
FUNCTION "FC_AI_MAPPING" : VOID
TITLE =
VERSION : 0.1


VAR_TEMP
  PIW512_DI : DINT ;
END_VAR
BEGIN

NETWORK
TITLE =
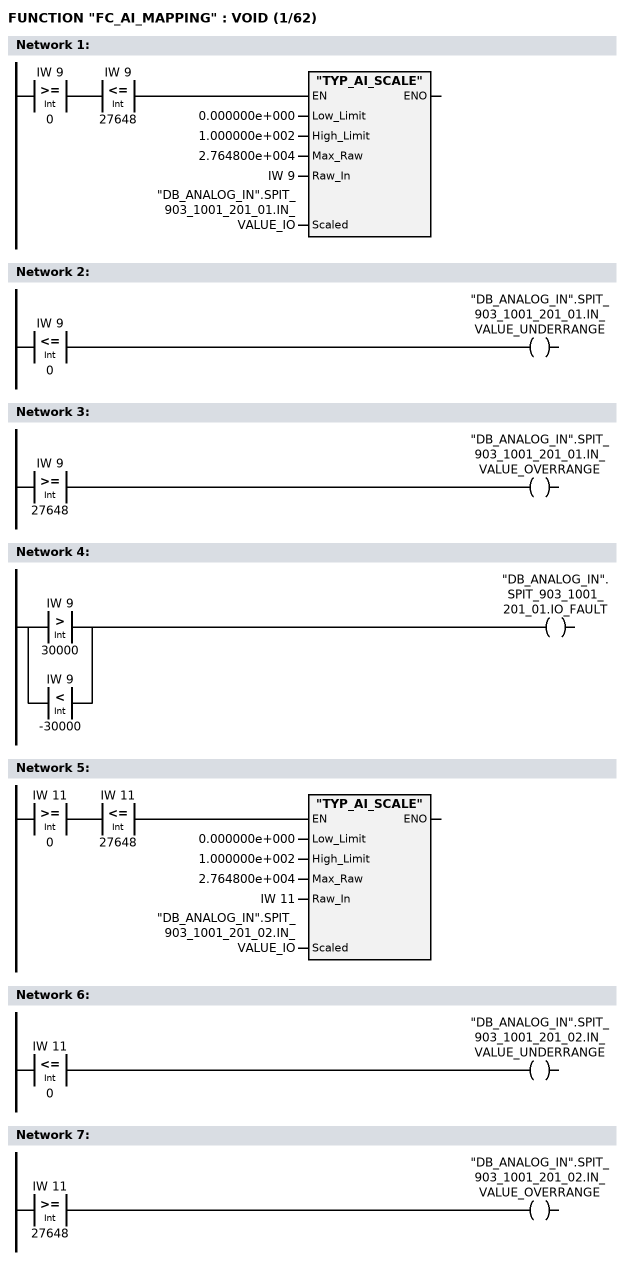

      A(    ;
      L     IW      9;
      L     0;
      >=I   ;
      )     ;
      A(    ;
      L     IW      9;

      L     27648;
      <=I   ;
      )     ;
      JNB   _001;
      CALL "TYP_AI_SCALE" (
           Low_Limit                := 0.000000e+000,
           High_Limit               := 1.000000e+002,
           Max_Raw                  := 2.764800e+004,
           Raw_In                   := IW      9,
           Scaled                   := "DB_ANALOG_IN".SPIT_903_1001_201_01.IN_VALUE_IO);
_001: NOP   0;
NETWORK
TITLE =

      L     IW      9;
      L     0;
      <=I   ;
      =     "DB_ANALOG_IN".SPIT_903_1001_201_01.IN_VALUE_UNDERRANGE;
NETWORK
TITLE =

      L     IW      9;
      L     27648;
      >=I   ;
      =     "DB_ANALOG_IN".SPIT_903_1001_201_01.IN_VALUE_OVERRANGE;
NETWORK
TITLE =

      O(    ;
      L     IW      9;
      L     30000;
      >I    ;
      )     ;
      O(    ;
      L     IW      9;
      L     -30000;
      <I    ;
      )     ;
      =     "DB_ANALOG_IN".SPIT_903_1001_201_01.IO_FAULT;

NETWORK
TITLE =

      A(    ;
      L     IW      11;
      L     0;
      >=I   ;
      )     ;
      A(    ;
      L     IW      11;

      L     27648;
      <=I   ;
      )     ;
      JNB   _002;
      CALL "TYP_AI_SCALE" (
           Low_Limit                := 0.000000e+000,
           High_Limit               := 1.000000e+002,
           Max_Raw                  := 2.764800e+004,
           Raw_In                   := IW      11,
           Scaled                   := "DB_ANALOG_IN".SPIT_903_1001_201_02.IN_VALUE_IO);
_002: NOP   0;
NETWORK
TITLE =

      L     IW      11;
      L     0;
      <=I   ;
      =     "DB_ANALOG_IN".SPIT_903_1001_201_02.IN_VALUE_UNDERRANGE;
NETWORK
TITLE =

      L     IW      11;
      L     27648;
      >=I   ;
      =     "DB_ANALOG_IN".SPIT_903_1001_201_02.IN_VALUE_OVERRANGE;
NETWORK
TITLE =
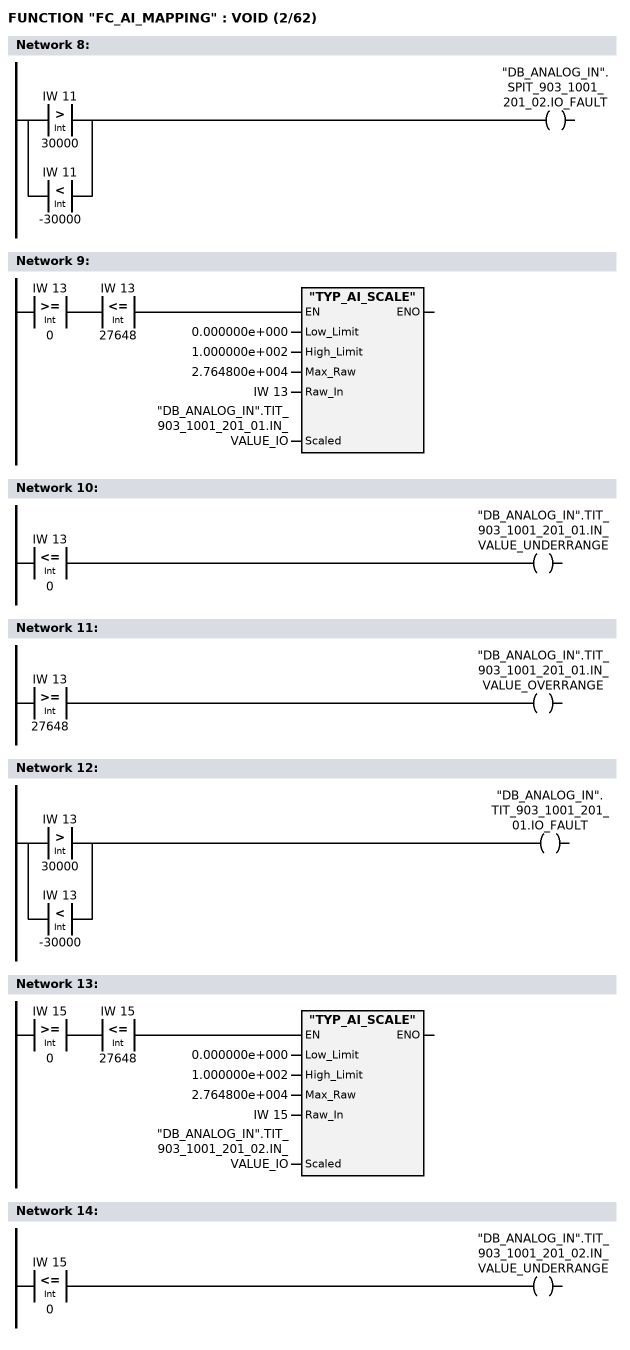

      O(    ;
      L     IW      11;
      L     30000;
      >I    ;
      )     ;
      O(    ;
      L     IW      11;
      L     -30000;
      <I    ;
      )     ;
      =     "DB_ANALOG_IN".SPIT_903_1001_201_02.IO_FAULT;

NETWORK
TITLE =

      A(    ;
      L     IW      13;
      L     0;
      >=I   ;
      )     ;
      A(    ;
      L     IW      13;

      L     27648;
      <=I   ;
      )     ;
      JNB   _003;
      CALL "TYP_AI_SCALE" (
           Low_Limit                := 0.000000e+000,
           High_Limit               := 1.000000e+002,
           Max_Raw                  := 2.764800e+004,
           Raw_In                   := IW      13,
           Scaled                   := "DB_ANALOG_IN".TIT_903_1001_201_01.IN_VALUE_IO);
_003: NOP   0;
NETWORK
TITLE =

      L     IW      13;
      L     0;
      <=I   ;
      =     "DB_ANALOG_IN".TIT_903_1001_201_01.IN_VALUE_UNDERRANGE;
NETWORK
TITLE =

      L     IW      13;
      L     27648;
      >=I   ;
      =     "DB_ANALOG_IN".TIT_903_1001_201_01.IN_VALUE_OVERRANGE;
NETWORK
TITLE =

      O(    ;
      L     IW      13;
      L     30000;
      >I    ;
      )     ;
      O(    ;
      L     IW      13;
      L     -30000;
      <I    ;
      )     ;
      =     "DB_ANALOG_IN".TIT_903_1001_201_01.IO_FAULT;

NETWORK
TITLE =

      A(    ;
      L     IW      15;
      L     0;
      >=I   ;
      )     ;
      A(    ;
      L     IW      15;

      L     27648;
      <=I   ;
      )     ;
      JNB   _004;
      CALL "TYP_AI_SCALE" (
           Low_Limit                := 0.000000e+000,
           High_Limit               := 1.000000e+002,
           Max_Raw                  := 2.764800e+004,
           Raw_In                   := IW      15,
           Scaled                   := "DB_ANALOG_IN".TIT_903_1001_201_02.IN_VALUE_IO);
_004: NOP   0;
NETWORK
TITLE =

      L     IW      15;
      L     0;
      <=I   ;
      =     "DB_ANALOG_IN".TIT_903_1001_201_02.IN_VALUE_UNDERRANGE;
NETWORK
TITLE =
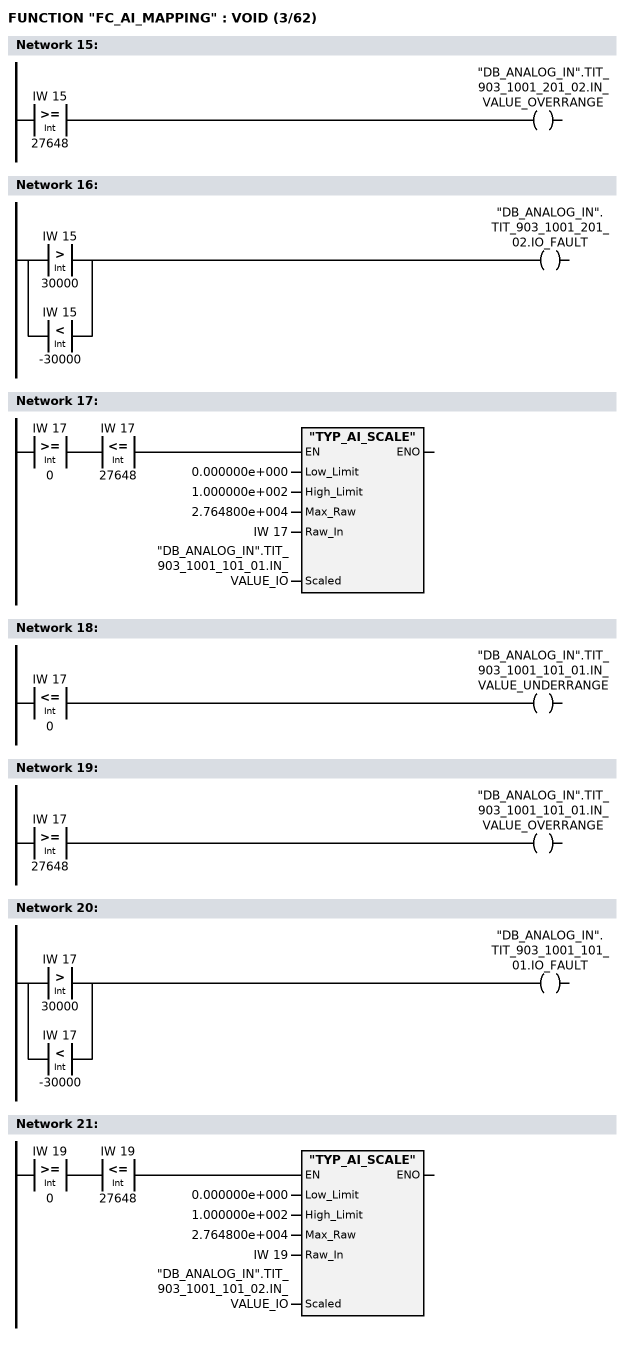

      L     IW      15;
      L     27648;
      >=I   ;
      =     "DB_ANALOG_IN".TIT_903_1001_201_02.IN_VALUE_OVERRANGE;
NETWORK
TITLE =

      O(    ;
      L     IW      15;
      L     30000;
      >I    ;
      )     ;
      O(    ;
      L     IW      15;
      L     -30000;
      <I    ;
      )     ;
      =     "DB_ANALOG_IN".TIT_903_1001_201_02.IO_FAULT;

NETWORK
TITLE =

      A(    ;
      L     IW      17;
      L     0;
      >=I   ;
      )     ;
      A(    ;
      L     IW      17;

      L     27648;
      <=I   ;
      )     ;
      JNB   _005;
      CALL "TYP_AI_SCALE" (
           Low_Limit                := 0.000000e+000,
           High_Limit               := 1.000000e+002,
           Max_Raw                  := 2.764800e+004,
           Raw_In                   := IW      17,
           Scaled                   := "DB_ANALOG_IN".TIT_903_1001_101_01.IN_VALUE_IO);
_005: NOP   0;
NETWORK
TITLE =

      L     IW      17;
      L     0;
      <=I   ;
      =     "DB_ANALOG_IN".TIT_903_1001_101_01.IN_VALUE_UNDERRANGE;
NETWORK
TITLE =

      L     IW      17;
      L     27648;
      >=I   ;
      =     "DB_ANALOG_IN".TIT_903_1001_101_01.IN_VALUE_OVERRANGE;
NETWORK
TITLE =

      O(    ;
      L     IW      17;
      L     30000;
      >I    ;
      )     ;
      O(    ;
      L     IW      17;
      L     -30000;
      <I    ;
      )     ;
      =     "DB_ANALOG_IN".TIT_903_1001_101_01.IO_FAULT;

NETWORK
TITLE =

      A(    ;
      L     IW      19;
      L     0;
      >=I   ;
      )     ;
      A(    ;
      L     IW      19;

      L     27648;
      <=I   ;
      )     ;
      JNB   _006;
      CALL "TYP_AI_SCALE" (
           Low_Limit                := 0.000000e+000,
           High_Limit               := 1.000000e+002,
           Max_Raw                  := 2.764800e+004,
           Raw_In                   := IW      19,
           Scaled                   := "DB_ANALOG_IN".TIT_903_1001_101_02.IN_VALUE_IO);
_006: NOP   0;
NETWORK
TITLE =
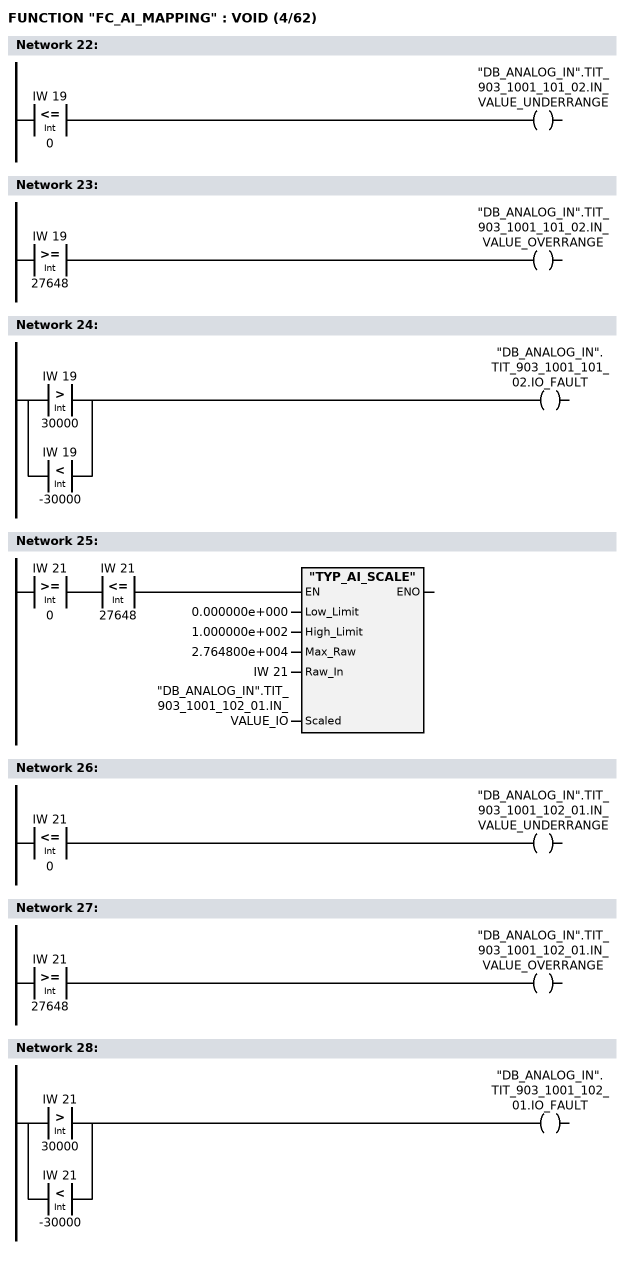

      L     IW      19;
      L     0;
      <=I   ;
      =     "DB_ANALOG_IN".TIT_903_1001_101_02.IN_VALUE_UNDERRANGE;
NETWORK
TITLE =

      L     IW      19;
      L     27648;
      >=I   ;
      =     "DB_ANALOG_IN".TIT_903_1001_101_02.IN_VALUE_OVERRANGE;
NETWORK
TITLE =

      O(    ;
      L     IW      19;
      L     30000;
      >I    ;
      )     ;
      O(    ;
      L     IW      19;
      L     -30000;
      <I    ;
      )     ;
      =     "DB_ANALOG_IN".TIT_903_1001_101_02.IO_FAULT;

NETWORK
TITLE =

      A(    ;
      L     IW      21;
      L     0;
      >=I   ;
      )     ;
      A(    ;
      L     IW      21;

      L     27648;
      <=I   ;
      )     ;
      JNB   _007;
      CALL "TYP_AI_SCALE" (
           Low_Limit                := 0.000000e+000,
           High_Limit               := 1.000000e+002,
           Max_Raw                  := 2.764800e+004,
           Raw_In                   := IW      21,
           Scaled                   := "DB_ANALOG_IN".TIT_903_1001_102_01.IN_VALUE_IO);
_007: NOP   0;
NETWORK
TITLE =

      L     IW      21;
      L     0;
      <=I   ;
      =     "DB_ANALOG_IN".TIT_903_1001_102_01.IN_VALUE_UNDERRANGE;
NETWORK
TITLE =

      L     IW      21;
      L     27648;
      >=I   ;
      =     "DB_ANALOG_IN".TIT_903_1001_102_01.IN_VALUE_OVERRANGE;
NETWORK
TITLE =

      O(    ;
      L     IW      21;
      L     30000;
      >I    ;
      )     ;
      O(    ;
      L     IW      21;
      L     -30000;
      <I    ;
      )     ;
      =     "DB_ANALOG_IN".TIT_903_1001_102_01.IO_FAULT;

NETWORK
TITLE =
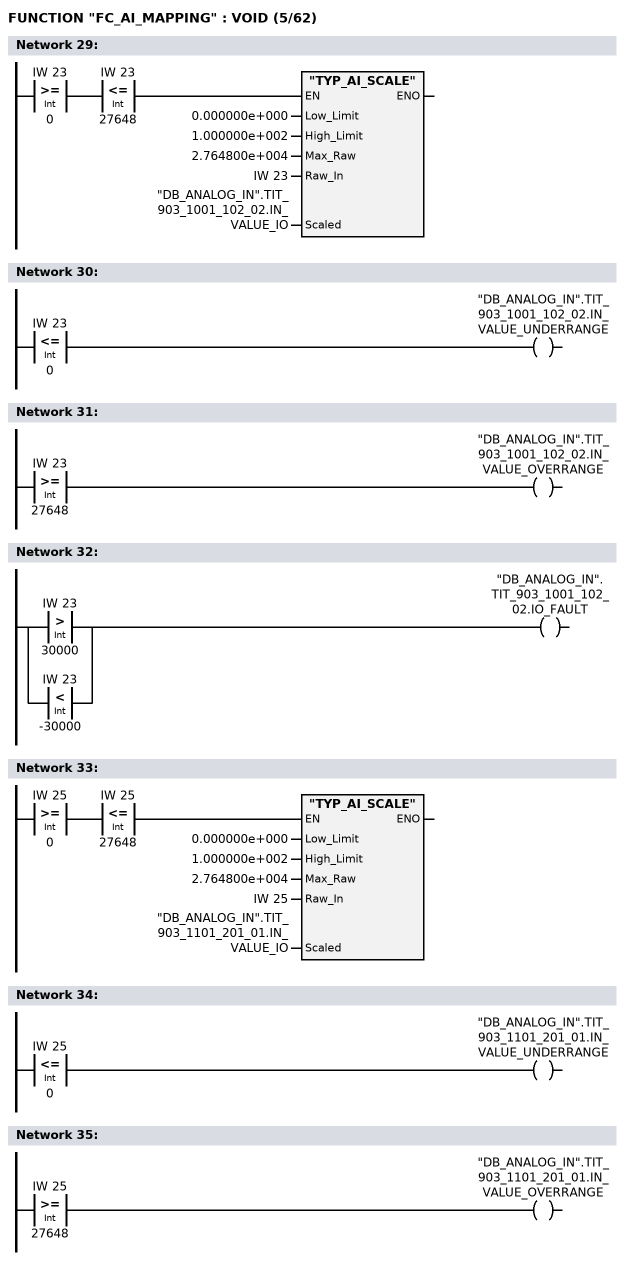

      A(    ;
      L     IW      23;
      L     0;
      >=I   ;
      )     ;
      A(    ;
      L     IW      23;

      L     27648;
      <=I   ;
      )     ;
      JNB   _008;
      CALL "TYP_AI_SCALE" (
           Low_Limit                := 0.000000e+000,
           High_Limit               := 1.000000e+002,
           Max_Raw                  := 2.764800e+004,
           Raw_In                   := IW      23,
           Scaled                   := "DB_ANALOG_IN".TIT_903_1001_102_02.IN_VALUE_IO);
_008: NOP   0;
NETWORK
TITLE =

      L     IW      23;
      L     0;
      <=I   ;
      =     "DB_ANALOG_IN".TIT_903_1001_102_02.IN_VALUE_UNDERRANGE;
NETWORK
TITLE =

      L     IW      23;
      L     27648;
      >=I   ;
      =     "DB_ANALOG_IN".TIT_903_1001_102_02.IN_VALUE_OVERRANGE;
NETWORK
TITLE =

      O(    ;
      L     IW      23;
      L     30000;
      >I    ;
      )     ;
      O(    ;
      L     IW      23;
      L     -30000;
      <I    ;
      )     ;
      =     "DB_ANALOG_IN".TIT_903_1001_102_02.IO_FAULT;

NETWORK
TITLE =

      A(    ;
      L     IW      25;
      L     0;
      >=I   ;
      )     ;
      A(    ;
      L     IW      25;

      L     27648;
      <=I   ;
      )     ;
      JNB   _009;
      CALL "TYP_AI_SCALE" (
           Low_Limit                := 0.000000e+000,
           High_Limit               := 1.000000e+002,
           Max_Raw                  := 2.764800e+004,
           Raw_In                   := IW      25,
           Scaled                   := "DB_ANALOG_IN".TIT_903_1101_201_01.IN_VALUE_IO);
_009: NOP   0;
NETWORK
TITLE =

      L     IW      25;
      L     0;
      <=I   ;
      =     "DB_ANALOG_IN".TIT_903_1101_201_01.IN_VALUE_UNDERRANGE;
NETWORK
TITLE =

      L     IW      25;
      L     27648;
      >=I   ;
      =     "DB_ANALOG_IN".TIT_903_1101_201_01.IN_VALUE_OVERRANGE;
NETWORK
TITLE =
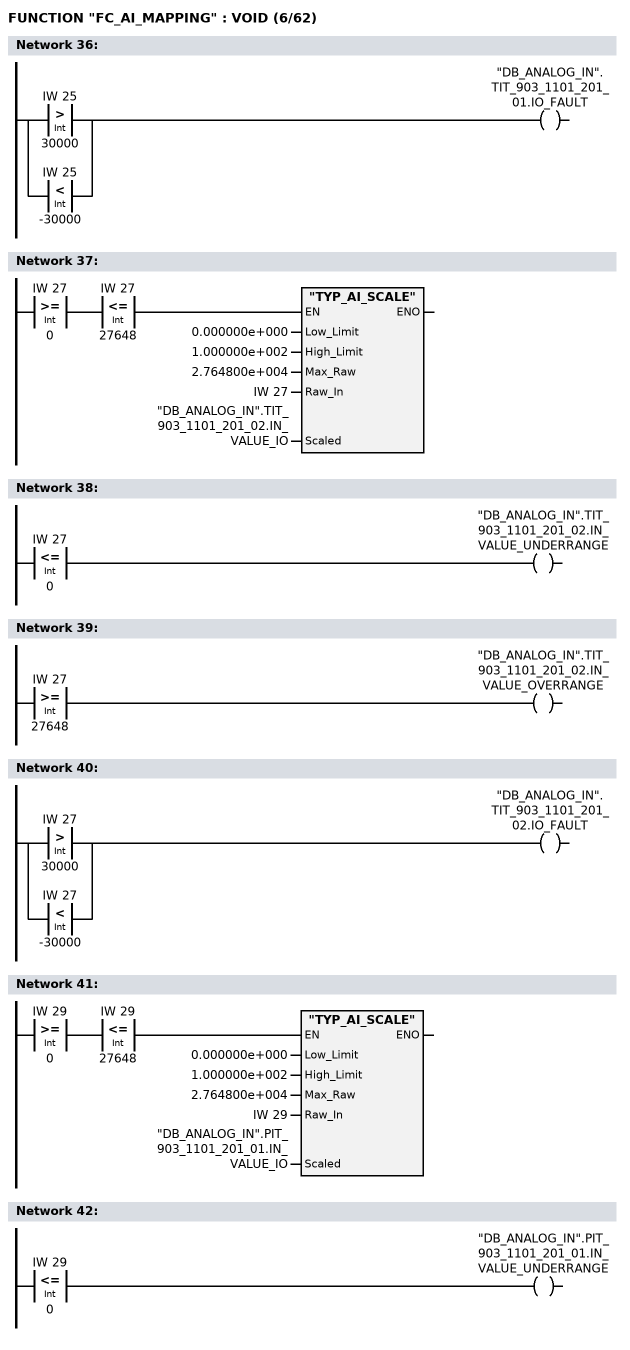

      O(    ;
      L     IW      25;
      L     30000;
      >I    ;
      )     ;
      O(    ;
      L     IW      25;
      L     -30000;
      <I    ;
      )     ;
      =     "DB_ANALOG_IN".TIT_903_1101_201_01.IO_FAULT;

NETWORK
TITLE =

      A(    ;
      L     IW      27;
      L     0;
      >=I   ;
      )     ;
      A(    ;
      L     IW      27;

      L     27648;
      <=I   ;
      )     ;
      JNB   _00a;
      CALL "TYP_AI_SCALE" (
           Low_Limit                := 0.000000e+000,
           High_Limit               := 1.000000e+002,
           Max_Raw                  := 2.764800e+004,
           Raw_In                   := IW      27,
           Scaled                   := "DB_ANALOG_IN".TIT_903_1101_201_02.IN_VALUE_IO);
_00a: NOP   0;
NETWORK
TITLE =

      L     IW      27;
      L     0;
      <=I   ;
      =     "DB_ANALOG_IN".TIT_903_1101_201_02.IN_VALUE_UNDERRANGE;
NETWORK
TITLE =

      L     IW      27;
      L     27648;
      >=I   ;
      =     "DB_ANALOG_IN".TIT_903_1101_201_02.IN_VALUE_OVERRANGE;
NETWORK
TITLE =

      O(    ;
      L     IW      27;
      L     30000;
      >I    ;
      )     ;
      O(    ;
      L     IW      27;
      L     -30000;
      <I    ;
      )     ;
      =     "DB_ANALOG_IN".TIT_903_1101_201_02.IO_FAULT;

NETWORK
TITLE =

      A(    ;
      L     IW      29;
      L     0;
      >=I   ;
      )     ;
      A(    ;
      L     IW      29;

      L     27648;
      <=I   ;
      )     ;
      JNB   _00b;
      CALL "TYP_AI_SCALE" (
           Low_Limit                := 0.000000e+000,
           High_Limit               := 1.000000e+002,
           Max_Raw                  := 2.764800e+004,
           Raw_In                   := IW      29,
           Scaled                   := "DB_ANALOG_IN".PIT_903_1101_201_01.IN_VALUE_IO);
_00b: NOP   0;
NETWORK
TITLE =

      L     IW      29;
      L     0;
      <=I   ;
      =     "DB_ANALOG_IN".PIT_903_1101_201_01.IN_VALUE_UNDERRANGE;
NETWORK
TITLE =
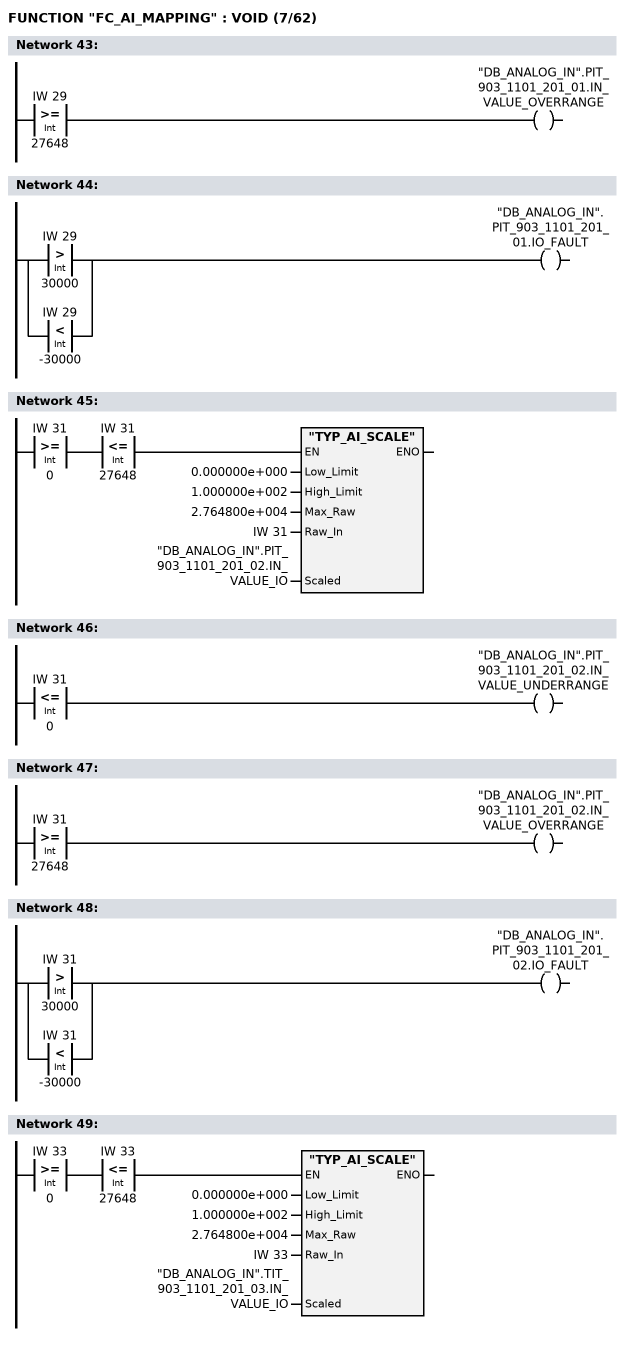

      L     IW      29;
      L     27648;
      >=I   ;
      =     "DB_ANALOG_IN".PIT_903_1101_201_01.IN_VALUE_OVERRANGE;
NETWORK
TITLE =

      O(    ;
      L     IW      29;
      L     30000;
      >I    ;
      )     ;
      O(    ;
      L     IW      29;
      L     -30000;
      <I    ;
      )     ;
      =     "DB_ANALOG_IN".PIT_903_1101_201_01.IO_FAULT;

NETWORK
TITLE =

      A(    ;
      L     IW      31;
      L     0;
      >=I   ;
      )     ;
      A(    ;
      L     IW      31;

      L     27648;
      <=I   ;
      )     ;
      JNB   _00c;
      CALL "TYP_AI_SCALE" (
           Low_Limit                := 0.000000e+000,
           High_Limit               := 1.000000e+002,
           Max_Raw                  := 2.764800e+004,
           Raw_In                   := IW      31,
           Scaled                   := "DB_ANALOG_IN".PIT_903_1101_201_02.IN_VALUE_IO);
_00c: NOP   0;
NETWORK
TITLE =

      L     IW      31;
      L     0;
      <=I   ;
      =     "DB_ANALOG_IN".PIT_903_1101_201_02.IN_VALUE_UNDERRANGE;
NETWORK
TITLE =

      L     IW      31;
      L     27648;
      >=I   ;
      =     "DB_ANALOG_IN".PIT_903_1101_201_02.IN_VALUE_OVERRANGE;
NETWORK
TITLE =

      O(    ;
      L     IW      31;
      L     30000;
      >I    ;
      )     ;
      O(    ;
      L     IW      31;
      L     -30000;
      <I    ;
      )     ;
      =     "DB_ANALOG_IN".PIT_903_1101_201_02.IO_FAULT;

NETWORK
TITLE =

      A(    ;
      L     IW      33;
      L     0;
      >=I   ;
      )     ;
      A(    ;
      L     IW      33;

      L     27648;
      <=I   ;
      )     ;
      JNB   _00d;
      CALL "TYP_AI_SCALE" (
           Low_Limit                := 0.000000e+000,
           High_Limit               := 1.000000e+002,
           Max_Raw                  := 2.764800e+004,
           Raw_In                   := IW      33,
           Scaled                   := "DB_ANALOG_IN".TIT_903_1101_201_03.IN_VALUE_IO);
_00d: NOP   0;
NETWORK
TITLE =
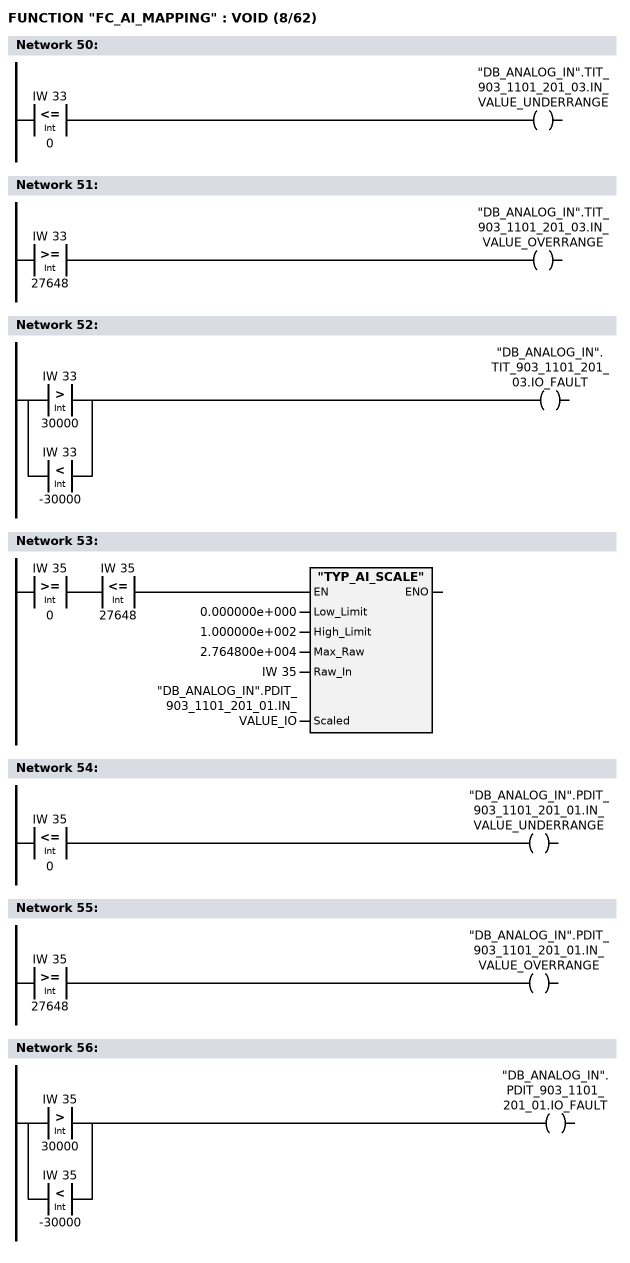

      L     IW      33;
      L     0;
      <=I   ;
      =     "DB_ANALOG_IN".TIT_903_1101_201_03.IN_VALUE_UNDERRANGE;
NETWORK
TITLE =

      L     IW      33;
      L     27648;
      >=I   ;
      =     "DB_ANALOG_IN".TIT_903_1101_201_03.IN_VALUE_OVERRANGE;
NETWORK
TITLE =

      O(    ;
      L     IW      33;
      L     30000;
      >I    ;
      )     ;
      O(    ;
      L     IW      33;
      L     -30000;
      <I    ;
      )     ;
      =     "DB_ANALOG_IN".TIT_903_1101_201_03.IO_FAULT;

NETWORK
TITLE =

      A(    ;
      L     IW      35;
      L     0;
      >=I   ;
      )     ;
      A(    ;
      L     IW      35;

      L     27648;
      <=I   ;
      )     ;
      JNB   _00e;
      CALL "TYP_AI_SCALE" (
           Low_Limit                := 0.000000e+000,
           High_Limit               := 1.000000e+002,
           Max_Raw                  := 2.764800e+004,
           Raw_In                   := IW      35,
           Scaled                   := "DB_ANALOG_IN".PDIT_903_1101_201_01.IN_VALUE_IO);
_00e: NOP   0;
NETWORK
TITLE =

      L     IW      35;
      L     0;
      <=I   ;
      =     "DB_ANALOG_IN".PDIT_903_1101_201_01.IN_VALUE_UNDERRANGE;
NETWORK
TITLE =

      L     IW      35;
      L     27648;
      >=I   ;
      =     "DB_ANALOG_IN".PDIT_903_1101_201_01.IN_VALUE_OVERRANGE;
NETWORK
TITLE =

      O(    ;
      L     IW      35;
      L     30000;
      >I    ;
      )     ;
      O(    ;
      L     IW      35;
      L     -30000;
      <I    ;
      )     ;
      =     "DB_ANALOG_IN".PDIT_903_1101_201_01.IO_FAULT;

NETWORK
TITLE =
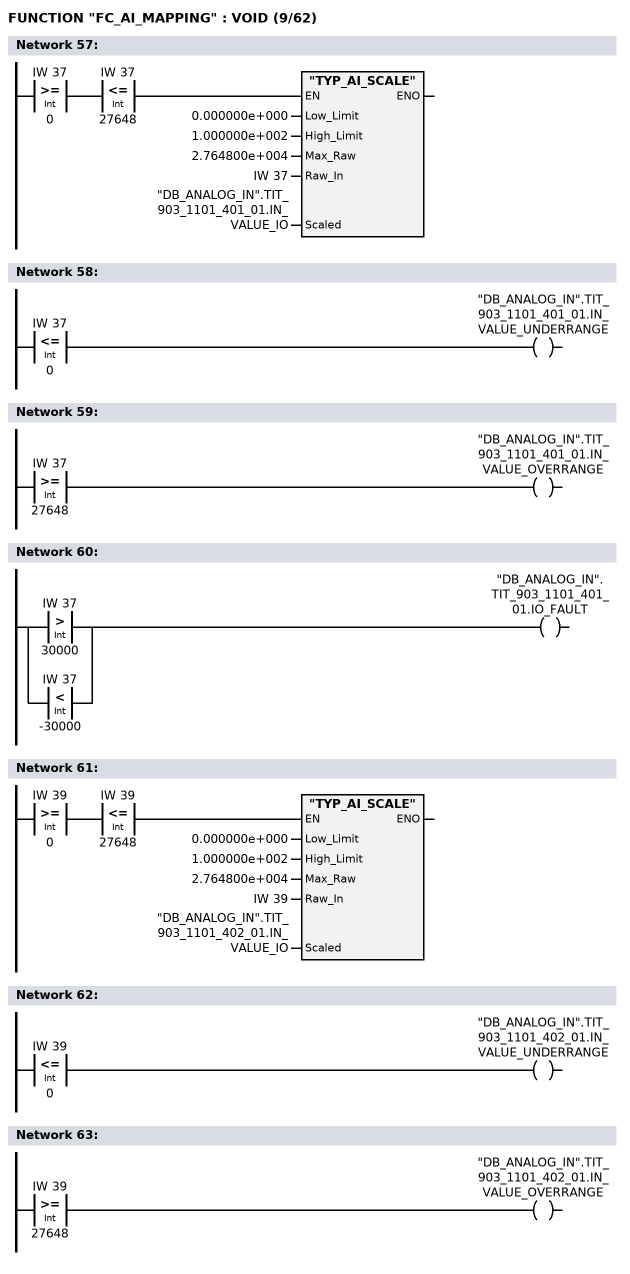

      A(    ;
      L     IW      37;
      L     0;
      >=I   ;
      )     ;
      A(    ;
      L     IW      37;

      L     27648;
      <=I   ;
      )     ;
      JNB   _00f;
      CALL "TYP_AI_SCALE" (
           Low_Limit                := 0.000000e+000,
           High_Limit               := 1.000000e+002,
           Max_Raw                  := 2.764800e+004,
           Raw_In                   := IW      37,
           Scaled                   := "DB_ANALOG_IN".TIT_903_1101_401_01.IN_VALUE_IO);
_00f: NOP   0;
NETWORK
TITLE =

      L     IW      37;
      L     0;
      <=I   ;
      =     "DB_ANALOG_IN".TIT_903_1101_401_01.IN_VALUE_UNDERRANGE;
NETWORK
TITLE =

      L     IW      37;
      L     27648;
      >=I   ;
      =     "DB_ANALOG_IN".TIT_903_1101_401_01.IN_VALUE_OVERRANGE;
NETWORK
TITLE =

      O(    ;
      L     IW      37;
      L     30000;
      >I    ;
      )     ;
      O(    ;
      L     IW      37;
      L     -30000;
      <I    ;
      )     ;
      =     "DB_ANALOG_IN".TIT_903_1101_401_01.IO_FAULT;

NETWORK
TITLE =

      A(    ;
      L     IW      39;
      L     0;
      >=I   ;
      )     ;
      A(    ;
      L     IW      39;

      L     27648;
      <=I   ;
      )     ;
      JNB   _010;
      CALL "TYP_AI_SCALE" (
           Low_Limit                := 0.000000e+000,
           High_Limit               := 1.000000e+002,
           Max_Raw                  := 2.764800e+004,
           Raw_In                   := IW      39,
           Scaled                   := "DB_ANALOG_IN".TIT_903_1101_402_01.IN_VALUE_IO);
_010: NOP   0;
NETWORK
TITLE =

      L     IW      39;
      L     0;
      <=I   ;
      =     "DB_ANALOG_IN".TIT_903_1101_402_01.IN_VALUE_UNDERRANGE;
NETWORK
TITLE =

      L     IW      39;
      L     27648;
      >=I   ;
      =     "DB_ANALOG_IN".TIT_903_1101_402_01.IN_VALUE_OVERRANGE;
NETWORK
TITLE =
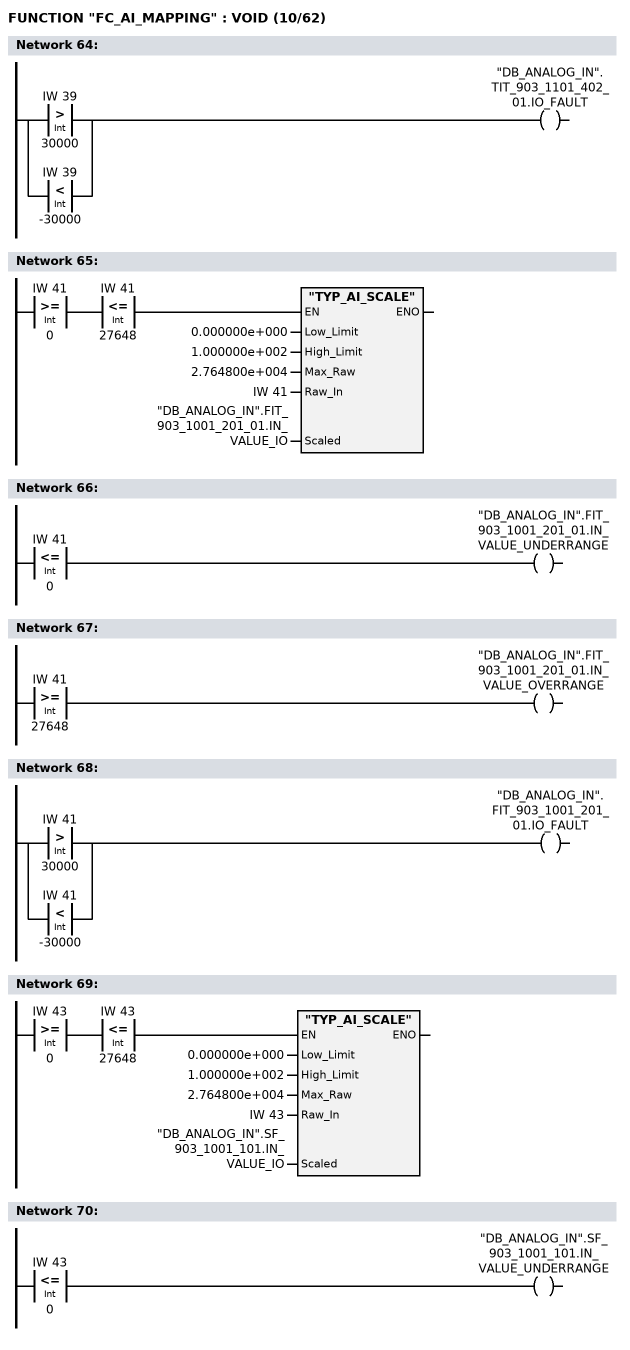

      O(    ;
      L     IW      39;
      L     30000;
      >I    ;
      )     ;
      O(    ;
      L     IW      39;
      L     -30000;
      <I    ;
      )     ;
      =     "DB_ANALOG_IN".TIT_903_1101_402_01.IO_FAULT;

NETWORK
TITLE =

      A(    ;
      L     IW      41;
      L     0;
      >=I   ;
      )     ;
      A(    ;
      L     IW      41;

      L     27648;
      <=I   ;
      )     ;
      JNB   _011;
      CALL "TYP_AI_SCALE" (
           Low_Limit                := 0.000000e+000,
           High_Limit               := 1.000000e+002,
           Max_Raw                  := 2.764800e+004,
           Raw_In                   := IW      41,
           Scaled                   := "DB_ANALOG_IN".FIT_903_1001_201_01.IN_VALUE_IO);
_011: NOP   0;
NETWORK
TITLE =

      L     IW      41;
      L     0;
      <=I   ;
      =     "DB_ANALOG_IN".FIT_903_1001_201_01.IN_VALUE_UNDERRANGE;
NETWORK
TITLE =

      L     IW      41;
      L     27648;
      >=I   ;
      =     "DB_ANALOG_IN".FIT_903_1001_201_01.IN_VALUE_OVERRANGE;
NETWORK
TITLE =

      O(    ;
      L     IW      41;
      L     30000;
      >I    ;
      )     ;
      O(    ;
      L     IW      41;
      L     -30000;
      <I    ;
      )     ;
      =     "DB_ANALOG_IN".FIT_903_1001_201_01.IO_FAULT;

NETWORK
TITLE =

      A(    ;
      L     IW      43;
      L     0;
      >=I   ;
      )     ;
      A(    ;
      L     IW      43;

      L     27648;
      <=I   ;
      )     ;
      JNB   _012;
      CALL "TYP_AI_SCALE" (
           Low_Limit                := 0.000000e+000,
           High_Limit               := 1.000000e+002,
           Max_Raw                  := 2.764800e+004,
           Raw_In                   := IW      43,
           Scaled                   := "DB_ANALOG_IN".SF_903_1001_101.IN_VALUE_IO);
_012: NOP   0;
NETWORK
TITLE =

      L     IW      43;
      L     0;
      <=I   ;
      =     "DB_ANALOG_IN".SF_903_1001_101.IN_VALUE_UNDERRANGE;
NETWORK
TITLE =
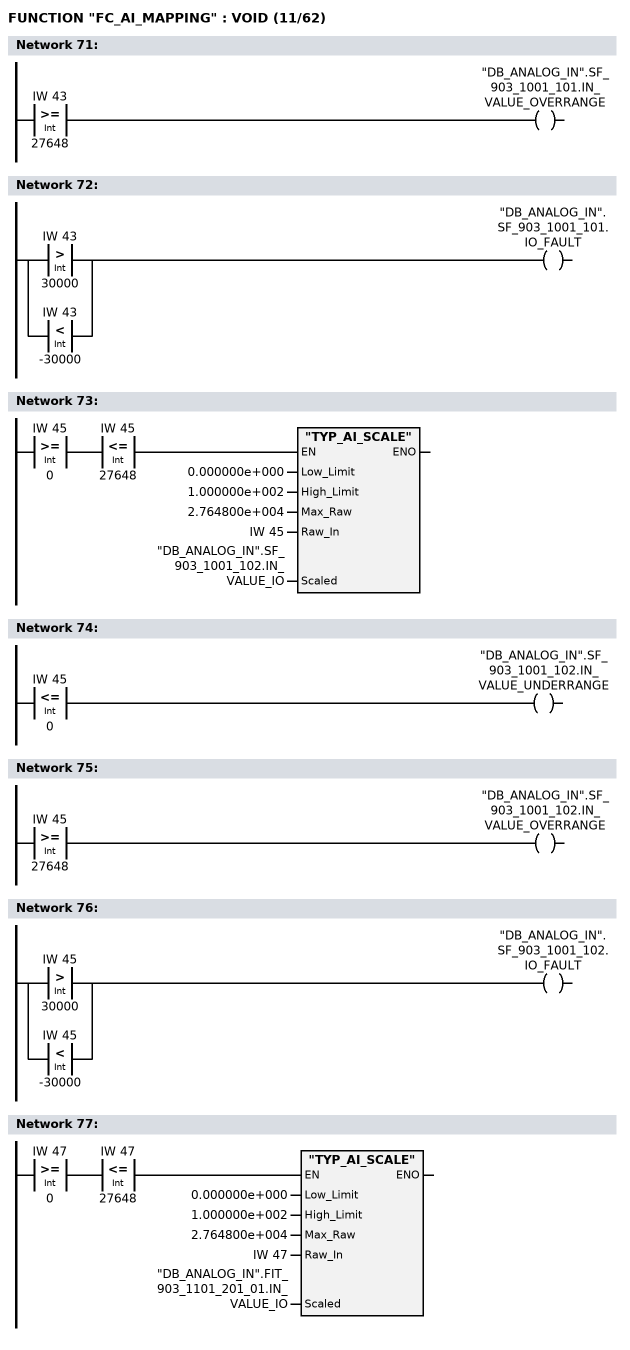

      L     IW      43;
      L     27648;
      >=I   ;
      =     "DB_ANALOG_IN".SF_903_1001_101.IN_VALUE_OVERRANGE;
NETWORK
TITLE =

      O(    ;
      L     IW      43;
      L     30000;
      >I    ;
      )     ;
      O(    ;
      L     IW      43;
      L     -30000;
      <I    ;
      )     ;
      =     "DB_ANALOG_IN".SF_903_1001_101.IO_FAULT;

NETWORK
TITLE =

      A(    ;
      L     IW      45;
      L     0;
      >=I   ;
      )     ;
      A(    ;
      L     IW      45;

      L     27648;
      <=I   ;
      )     ;
      JNB   _013;
      CALL "TYP_AI_SCALE" (
           Low_Limit                := 0.000000e+000,
           High_Limit               := 1.000000e+002,
           Max_Raw                  := 2.764800e+004,
           Raw_In                   := IW      45,
           Scaled                   := "DB_ANALOG_IN".SF_903_1001_102.IN_VALUE_IO);
_013: NOP   0;
NETWORK
TITLE =

      L     IW      45;
      L     0;
      <=I   ;
      =     "DB_ANALOG_IN".SF_903_1001_102.IN_VALUE_UNDERRANGE;
NETWORK
TITLE =

      L     IW      45;
      L     27648;
      >=I   ;
      =     "DB_ANALOG_IN".SF_903_1001_102.IN_VALUE_OVERRANGE;
NETWORK
TITLE =

      O(    ;
      L     IW      45;
      L     30000;
      >I    ;
      )     ;
      O(    ;
      L     IW      45;
      L     -30000;
      <I    ;
      )     ;
      =     "DB_ANALOG_IN".SF_903_1001_102.IO_FAULT;

NETWORK
TITLE =

      A(    ;
      L     IW      47;
      L     0;
      >=I   ;
      )     ;
      A(    ;
      L     IW      47;

      L     27648;
      <=I   ;
      )     ;
      JNB   _014;
      CALL "TYP_AI_SCALE" (
           Low_Limit                := 0.000000e+000,
           High_Limit               := 1.000000e+002,
           Max_Raw                  := 2.764800e+004,
           Raw_In                   := IW      47,
           Scaled                   := "DB_ANALOG_IN".FIT_903_1101_201_01.IN_VALUE_IO);
_014: NOP   0;
NETWORK
TITLE =
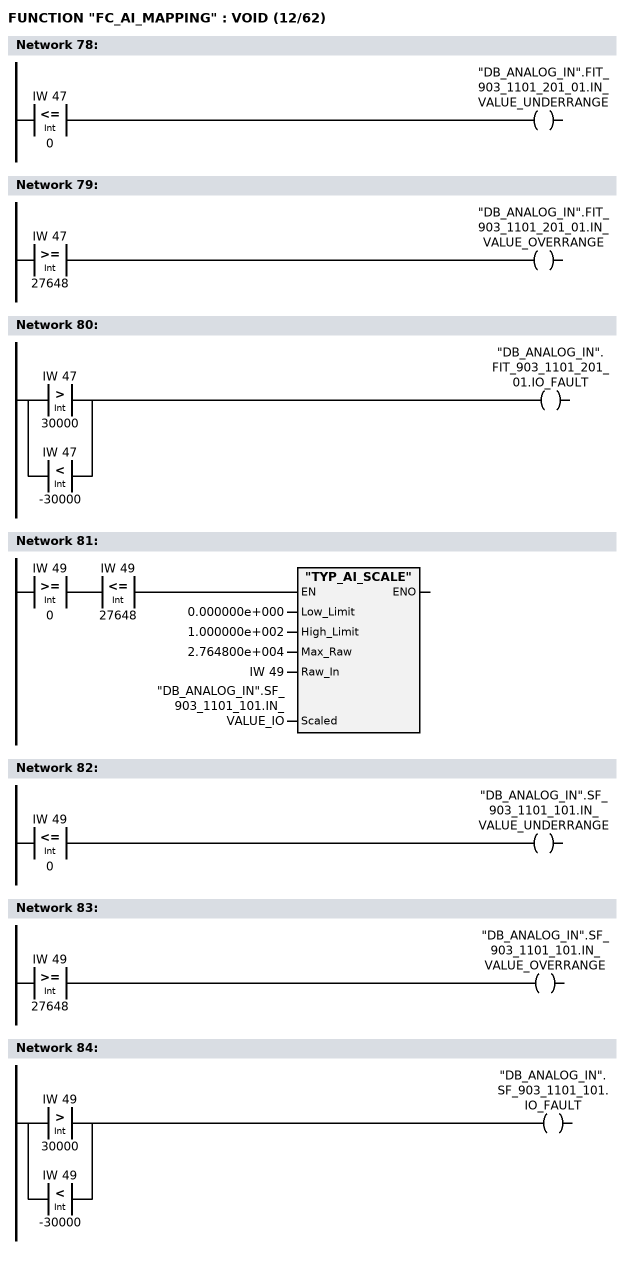

      L     IW      47;
      L     0;
      <=I   ;
      =     "DB_ANALOG_IN".FIT_903_1101_201_01.IN_VALUE_UNDERRANGE;
NETWORK
TITLE =

      L     IW      47;
      L     27648;
      >=I   ;
      =     "DB_ANALOG_IN".FIT_903_1101_201_01.IN_VALUE_OVERRANGE;
NETWORK
TITLE =

      O(    ;
      L     IW      47;
      L     30000;
      >I    ;
      )     ;
      O(    ;
      L     IW      47;
      L     -30000;
      <I    ;
      )     ;
      =     "DB_ANALOG_IN".FIT_903_1101_201_01.IO_FAULT;

NETWORK
TITLE =

      A(    ;
      L     IW      49;
      L     0;
      >=I   ;
      )     ;
      A(    ;
      L     IW      49;

      L     27648;
      <=I   ;
      )     ;
      JNB   _015;
      CALL "TYP_AI_SCALE" (
           Low_Limit                := 0.000000e+000,
           High_Limit               := 1.000000e+002,
           Max_Raw                  := 2.764800e+004,
           Raw_In                   := IW      49,
           Scaled                   := "DB_ANALOG_IN".SF_903_1101_101.IN_VALUE_IO);
_015: NOP   0;
NETWORK
TITLE =

      L     IW      49;
      L     0;
      <=I   ;
      =     "DB_ANALOG_IN".SF_903_1101_101.IN_VALUE_UNDERRANGE;
NETWORK
TITLE =

      L     IW      49;
      L     27648;
      >=I   ;
      =     "DB_ANALOG_IN".SF_903_1101_101.IN_VALUE_OVERRANGE;
NETWORK
TITLE =

      O(    ;
      L     IW      49;
      L     30000;
      >I    ;
      )     ;
      O(    ;
      L     IW      49;
      L     -30000;
      <I    ;
      )     ;
      =     "DB_ANALOG_IN".SF_903_1101_101.IO_FAULT;

NETWORK
TITLE =
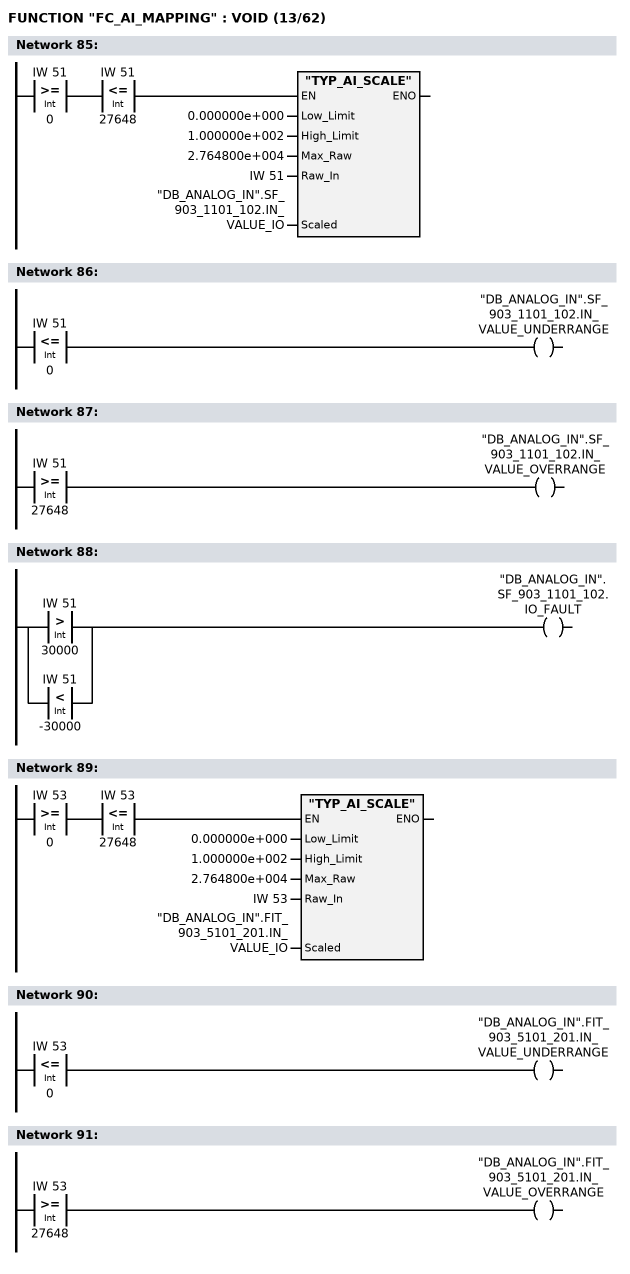

      A(    ;
      L     IW      51;
      L     0;
      >=I   ;
      )     ;
      A(    ;
      L     IW      51;

      L     27648;
      <=I   ;
      )     ;
      JNB   _016;
      CALL "TYP_AI_SCALE" (
           Low_Limit                := 0.000000e+000,
           High_Limit               := 1.000000e+002,
           Max_Raw                  := 2.764800e+004,
           Raw_In                   := IW      51,
           Scaled                   := "DB_ANALOG_IN".SF_903_1101_102.IN_VALUE_IO);
_016: NOP   0;
NETWORK
TITLE =

      L     IW      51;
      L     0;
      <=I   ;
      =     "DB_ANALOG_IN".SF_903_1101_102.IN_VALUE_UNDERRANGE;
NETWORK
TITLE =

      L     IW      51;
      L     27648;
      >=I   ;
      =     "DB_ANALOG_IN".SF_903_1101_102.IN_VALUE_OVERRANGE;
NETWORK
TITLE =

      O(    ;
      L     IW      51;
      L     30000;
      >I    ;
      )     ;
      O(    ;
      L     IW      51;
      L     -30000;
      <I    ;
      )     ;
      =     "DB_ANALOG_IN".SF_903_1101_102.IO_FAULT;

NETWORK
TITLE =

      A(    ;
      L     IW      53;
      L     0;
      >=I   ;
      )     ;
      A(    ;
      L     IW      53;

      L     27648;
      <=I   ;
      )     ;
      JNB   _017;
      CALL "TYP_AI_SCALE" (
           Low_Limit                := 0.000000e+000,
           High_Limit               := 1.000000e+002,
           Max_Raw                  := 2.764800e+004,
           Raw_In                   := IW      53,
           Scaled                   := "DB_ANALOG_IN".FIT_903_5101_201.IN_VALUE_IO);
_017: NOP   0;
NETWORK
TITLE =

      L     IW      53;
      L     0;
      <=I   ;
      =     "DB_ANALOG_IN".FIT_903_5101_201.IN_VALUE_UNDERRANGE;
NETWORK
TITLE =

      L     IW      53;
      L     27648;
      >=I   ;
      =     "DB_ANALOG_IN".FIT_903_5101_201.IN_VALUE_OVERRANGE;
NETWORK
TITLE =
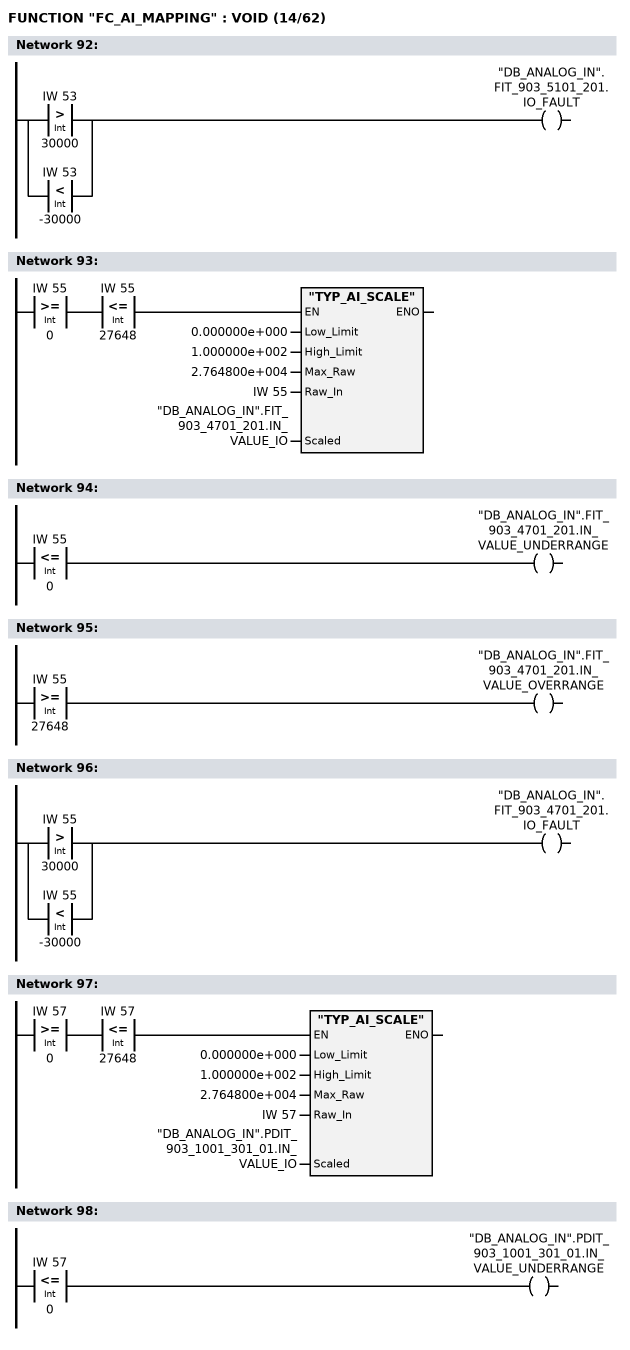

      O(    ;
      L     IW      53;
      L     30000;
      >I    ;
      )     ;
      O(    ;
      L     IW      53;
      L     -30000;
      <I    ;
      )     ;
      =     "DB_ANALOG_IN".FIT_903_5101_201.IO_FAULT;

NETWORK
TITLE =

      A(    ;
      L     IW      55;
      L     0;
      >=I   ;
      )     ;
      A(    ;
      L     IW      55;

      L     27648;
      <=I   ;
      )     ;
      JNB   _018;
      CALL "TYP_AI_SCALE" (
           Low_Limit                := 0.000000e+000,
           High_Limit               := 1.000000e+002,
           Max_Raw                  := 2.764800e+004,
           Raw_In                   := IW      55,
           Scaled                   := "DB_ANALOG_IN".FIT_903_4701_201.IN_VALUE_IO);
_018: NOP   0;
NETWORK
TITLE =

      L     IW      55;
      L     0;
      <=I   ;
      =     "DB_ANALOG_IN".FIT_903_4701_201.IN_VALUE_UNDERRANGE;
NETWORK
TITLE =

      L     IW      55;
      L     27648;
      >=I   ;
      =     "DB_ANALOG_IN".FIT_903_4701_201.IN_VALUE_OVERRANGE;
NETWORK
TITLE =

      O(    ;
      L     IW      55;
      L     30000;
      >I    ;
      )     ;
      O(    ;
      L     IW      55;
      L     -30000;
      <I    ;
      )     ;
      =     "DB_ANALOG_IN".FIT_903_4701_201.IO_FAULT;

NETWORK
TITLE =

      A(    ;
      L     IW      57;
      L     0;
      >=I   ;
      )     ;
      A(    ;
      L     IW      57;

      L     27648;
      <=I   ;
      )     ;
      JNB   _019;
      CALL "TYP_AI_SCALE" (
           Low_Limit                := 0.000000e+000,
           High_Limit               := 1.000000e+002,
           Max_Raw                  := 2.764800e+004,
           Raw_In                   := IW      57,
           Scaled                   := "DB_ANALOG_IN".PDIT_903_1001_301_01.IN_VALUE_IO);
_019: NOP   0;
NETWORK
TITLE =

      L     IW      57;
      L     0;
      <=I   ;
      =     "DB_ANALOG_IN".PDIT_903_1001_301_01.IN_VALUE_UNDERRANGE;
NETWORK
TITLE =
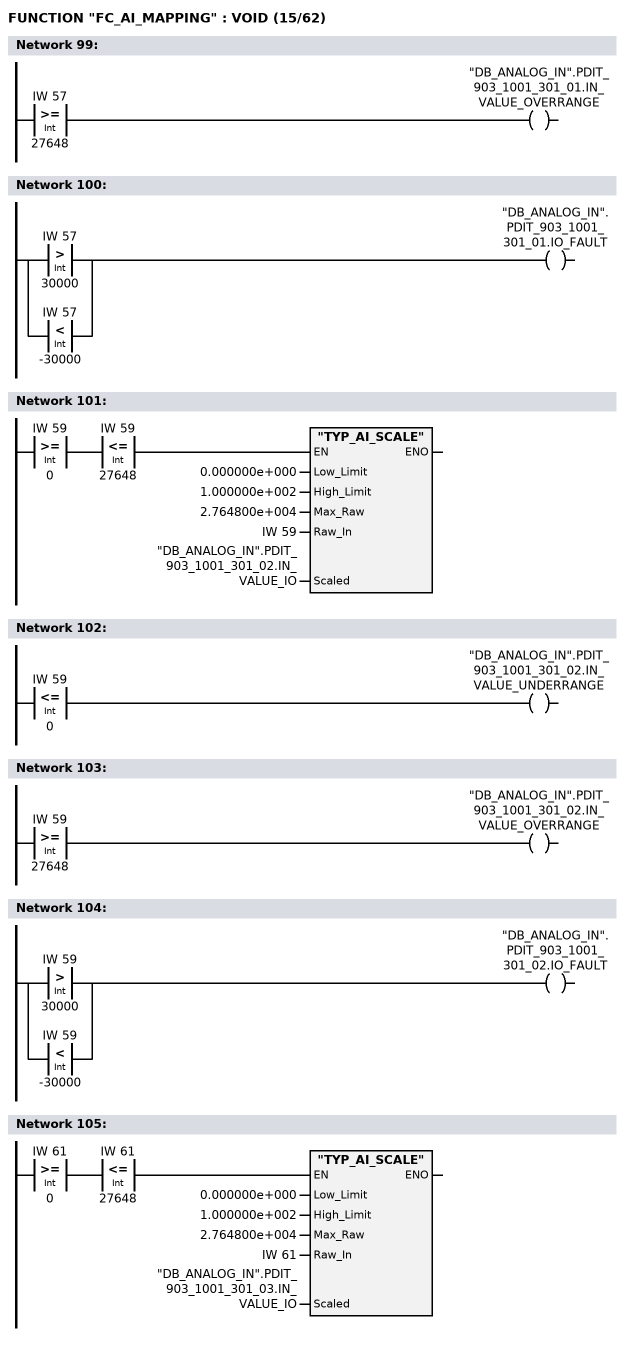

      L     IW      57;
      L     27648;
      >=I   ;
      =     "DB_ANALOG_IN".PDIT_903_1001_301_01.IN_VALUE_OVERRANGE;
NETWORK
TITLE =

      O(    ;
      L     IW      57;
      L     30000;
      >I    ;
      )     ;
      O(    ;
      L     IW      57;
      L     -30000;
      <I    ;
      )     ;
      =     "DB_ANALOG_IN".PDIT_903_1001_301_01.IO_FAULT;

NETWORK
TITLE =

      A(    ;
      L     IW      59;
      L     0;
      >=I   ;
      )     ;
      A(    ;
      L     IW      59;

      L     27648;
      <=I   ;
      )     ;
      JNB   _01a;
      CALL "TYP_AI_SCALE" (
           Low_Limit                := 0.000000e+000,
           High_Limit               := 1.000000e+002,
           Max_Raw                  := 2.764800e+004,
           Raw_In                   := IW      59,
           Scaled                   := "DB_ANALOG_IN".PDIT_903_1001_301_02.IN_VALUE_IO);
_01a: NOP   0;
NETWORK
TITLE =

      L     IW      59;
      L     0;
      <=I   ;
      =     "DB_ANALOG_IN".PDIT_903_1001_301_02.IN_VALUE_UNDERRANGE;
NETWORK
TITLE =

      L     IW      59;
      L     27648;
      >=I   ;
      =     "DB_ANALOG_IN".PDIT_903_1001_301_02.IN_VALUE_OVERRANGE;
NETWORK
TITLE =

      O(    ;
      L     IW      59;
      L     30000;
      >I    ;
      )     ;
      O(    ;
      L     IW      59;
      L     -30000;
      <I    ;
      )     ;
      =     "DB_ANALOG_IN".PDIT_903_1001_301_02.IO_FAULT;

NETWORK
TITLE =

      A(    ;
      L     IW      61;
      L     0;
      >=I   ;
      )     ;
      A(    ;
      L     IW      61;

      L     27648;
      <=I   ;
      )     ;
      JNB   _01b;
      CALL "TYP_AI_SCALE" (
           Low_Limit                := 0.000000e+000,
           High_Limit               := 1.000000e+002,
           Max_Raw                  := 2.764800e+004,
           Raw_In                   := IW      61,
           Scaled                   := "DB_ANALOG_IN".PDIT_903_1001_301_03.IN_VALUE_IO);
_01b: NOP   0;
NETWORK
TITLE =
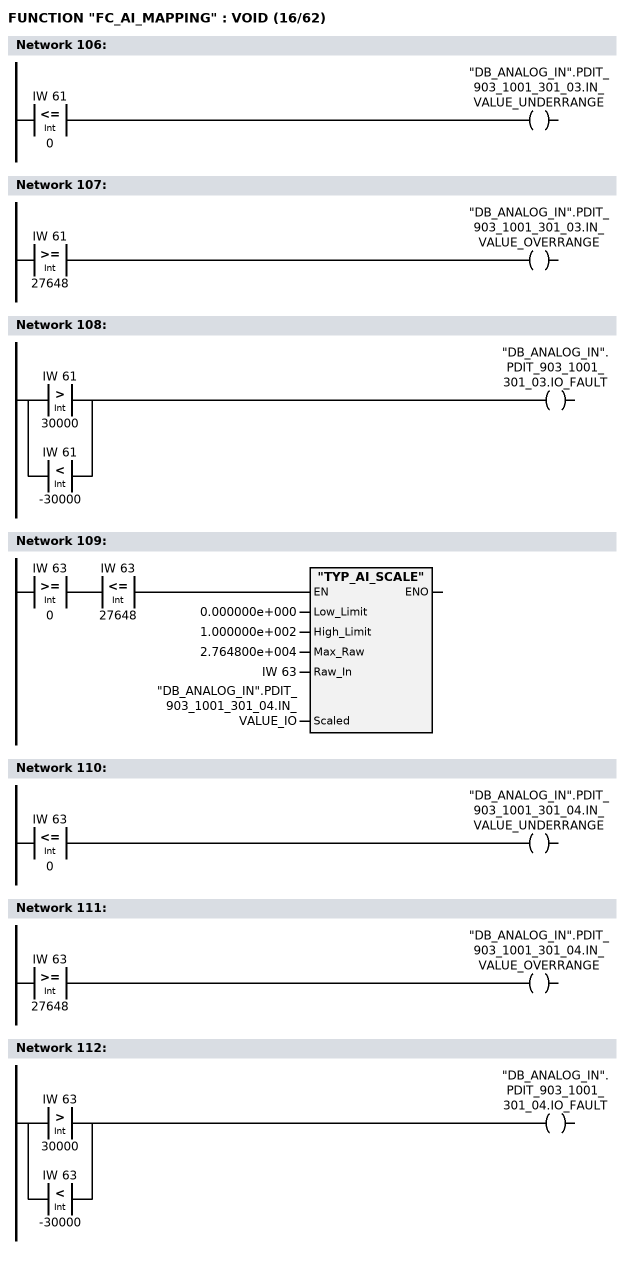

      L     IW      61;
      L     0;
      <=I   ;
      =     "DB_ANALOG_IN".PDIT_903_1001_301_03.IN_VALUE_UNDERRANGE;
NETWORK
TITLE =

      L     IW      61;
      L     27648;
      >=I   ;
      =     "DB_ANALOG_IN".PDIT_903_1001_301_03.IN_VALUE_OVERRANGE;
NETWORK
TITLE =

      O(    ;
      L     IW      61;
      L     30000;
      >I    ;
      )     ;
      O(    ;
      L     IW      61;
      L     -30000;
      <I    ;
      )     ;
      =     "DB_ANALOG_IN".PDIT_903_1001_301_03.IO_FAULT;

NETWORK
TITLE =

      A(    ;
      L     IW      63;
      L     0;
      >=I   ;
      )     ;
      A(    ;
      L     IW      63;

      L     27648;
      <=I   ;
      )     ;
      JNB   _01c;
      CALL "TYP_AI_SCALE" (
           Low_Limit                := 0.000000e+000,
           High_Limit               := 1.000000e+002,
           Max_Raw                  := 2.764800e+004,
           Raw_In                   := IW      63,
           Scaled                   := "DB_ANALOG_IN".PDIT_903_1001_301_04.IN_VALUE_IO);
_01c: NOP   0;
NETWORK
TITLE =

      L     IW      63;
      L     0;
      <=I   ;
      =     "DB_ANALOG_IN".PDIT_903_1001_301_04.IN_VALUE_UNDERRANGE;
NETWORK
TITLE =

      L     IW      63;
      L     27648;
      >=I   ;
      =     "DB_ANALOG_IN".PDIT_903_1001_301_04.IN_VALUE_OVERRANGE;
NETWORK
TITLE =

      O(    ;
      L     IW      63;
      L     30000;
      >I    ;
      )     ;
      O(    ;
      L     IW      63;
      L     -30000;
      <I    ;
      )     ;
      =     "DB_ANALOG_IN".PDIT_903_1001_301_04.IO_FAULT;

NETWORK
TITLE =
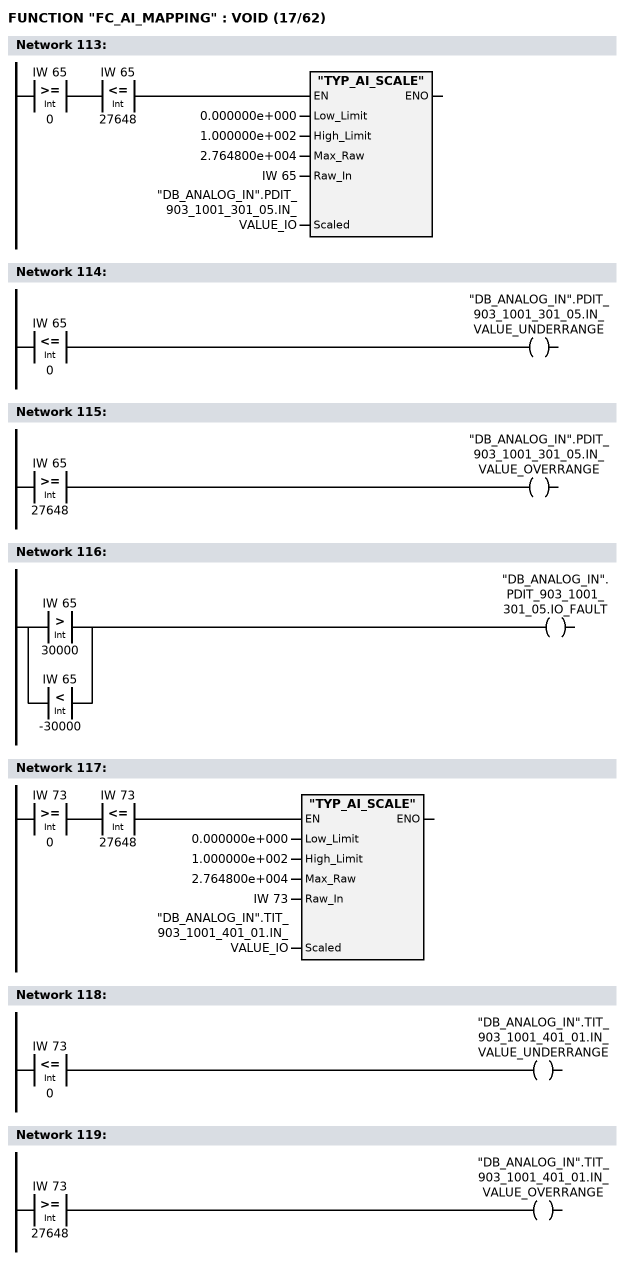

      A(    ;
      L     IW      65;
      L     0;
      >=I   ;
      )     ;
      A(    ;
      L     IW      65;

      L     27648;
      <=I   ;
      )     ;
      JNB   _01d;
      CALL "TYP_AI_SCALE" (
           Low_Limit                := 0.000000e+000,
           High_Limit               := 1.000000e+002,
           Max_Raw                  := 2.764800e+004,
           Raw_In                   := IW      65,
           Scaled                   := "DB_ANALOG_IN".PDIT_903_1001_301_05.IN_VALUE_IO);
_01d: NOP   0;
NETWORK
TITLE =

      L     IW      65;
      L     0;
      <=I   ;
      =     "DB_ANALOG_IN".PDIT_903_1001_301_05.IN_VALUE_UNDERRANGE;
NETWORK
TITLE =

      L     IW      65;
      L     27648;
      >=I   ;
      =     "DB_ANALOG_IN".PDIT_903_1001_301_05.IN_VALUE_OVERRANGE;
NETWORK
TITLE =

      O(    ;
      L     IW      65;
      L     30000;
      >I    ;
      )     ;
      O(    ;
      L     IW      65;
      L     -30000;
      <I    ;
      )     ;
      =     "DB_ANALOG_IN".PDIT_903_1001_301_05.IO_FAULT;

NETWORK
TITLE =

      A(    ;
      L     IW      73;
      L     0;
      >=I   ;
      )     ;
      A(    ;
      L     IW      73;

      L     27648;
      <=I   ;
      )     ;
      JNB   _01e;
      CALL "TYP_AI_SCALE" (
           Low_Limit                := 0.000000e+000,
           High_Limit               := 1.000000e+002,
           Max_Raw                  := 2.764800e+004,
           Raw_In                   := IW      73,
           Scaled                   := "DB_ANALOG_IN".TIT_903_1001_401_01.IN_VALUE_IO);
_01e: NOP   0;
NETWORK
TITLE =

      L     IW      73;
      L     0;
      <=I   ;
      =     "DB_ANALOG_IN".TIT_903_1001_401_01.IN_VALUE_UNDERRANGE;
NETWORK
TITLE =

      L     IW      73;
      L     27648;
      >=I   ;
      =     "DB_ANALOG_IN".TIT_903_1001_401_01.IN_VALUE_OVERRANGE;
NETWORK
TITLE =
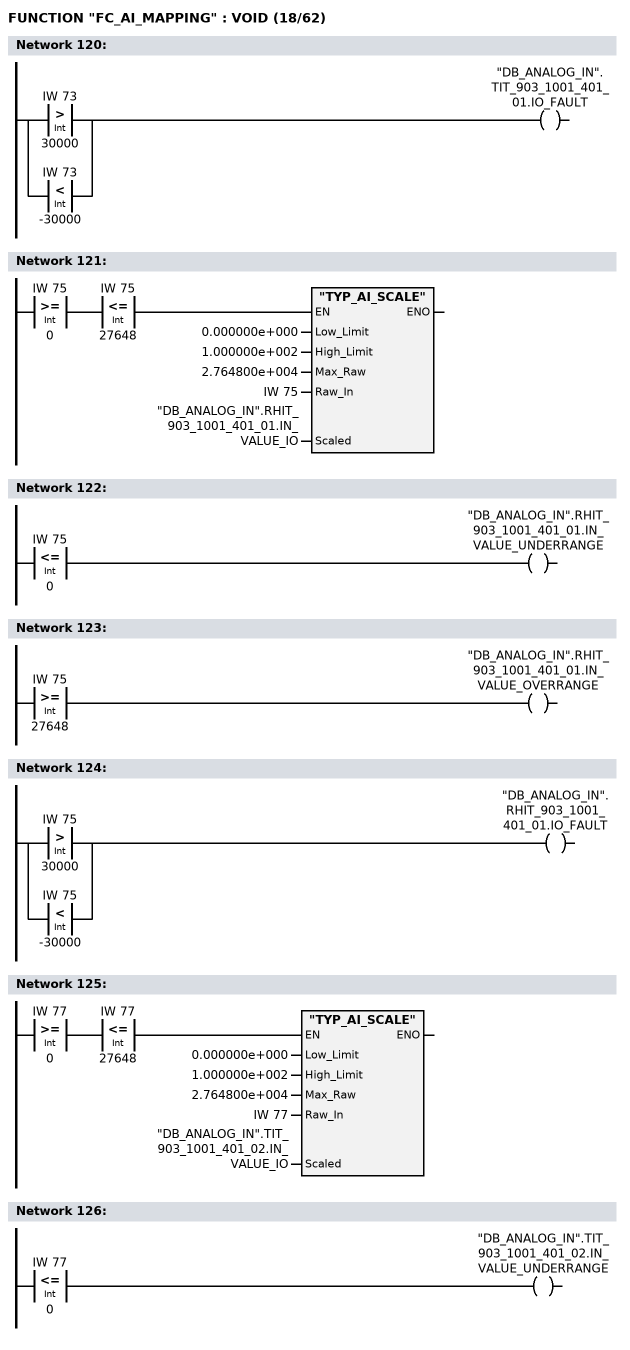

      O(    ;
      L     IW      73;
      L     30000;
      >I    ;
      )     ;
      O(    ;
      L     IW      73;
      L     -30000;
      <I    ;
      )     ;
      =     "DB_ANALOG_IN".TIT_903_1001_401_01.IO_FAULT;

NETWORK
TITLE =

      A(    ;
      L     IW      75;
      L     0;
      >=I   ;
      )     ;
      A(    ;
      L     IW      75;

      L     27648;
      <=I   ;
      )     ;
      JNB   _01f;
      CALL "TYP_AI_SCALE" (
           Low_Limit                := 0.000000e+000,
           High_Limit               := 1.000000e+002,
           Max_Raw                  := 2.764800e+004,
           Raw_In                   := IW      75,
           Scaled                   := "DB_ANALOG_IN".RHIT_903_1001_401_01.IN_VALUE_IO);
_01f: NOP   0;
NETWORK
TITLE =

      L     IW      75;
      L     0;
      <=I   ;
      =     "DB_ANALOG_IN".RHIT_903_1001_401_01.IN_VALUE_UNDERRANGE;
NETWORK
TITLE =

      L     IW      75;
      L     27648;
      >=I   ;
      =     "DB_ANALOG_IN".RHIT_903_1001_401_01.IN_VALUE_OVERRANGE;
NETWORK
TITLE =

      O(    ;
      L     IW      75;
      L     30000;
      >I    ;
      )     ;
      O(    ;
      L     IW      75;
      L     -30000;
      <I    ;
      )     ;
      =     "DB_ANALOG_IN".RHIT_903_1001_401_01.IO_FAULT;

NETWORK
TITLE =

      A(    ;
      L     IW      77;
      L     0;
      >=I   ;
      )     ;
      A(    ;
      L     IW      77;

      L     27648;
      <=I   ;
      )     ;
      JNB   _020;
      CALL "TYP_AI_SCALE" (
           Low_Limit                := 0.000000e+000,
           High_Limit               := 1.000000e+002,
           Max_Raw                  := 2.764800e+004,
           Raw_In                   := IW      77,
           Scaled                   := "DB_ANALOG_IN".TIT_903_1001_401_02.IN_VALUE_IO);
_020: NOP   0;
NETWORK
TITLE =

      L     IW      77;
      L     0;
      <=I   ;
      =     "DB_ANALOG_IN".TIT_903_1001_401_02.IN_VALUE_UNDERRANGE;
NETWORK
TITLE =
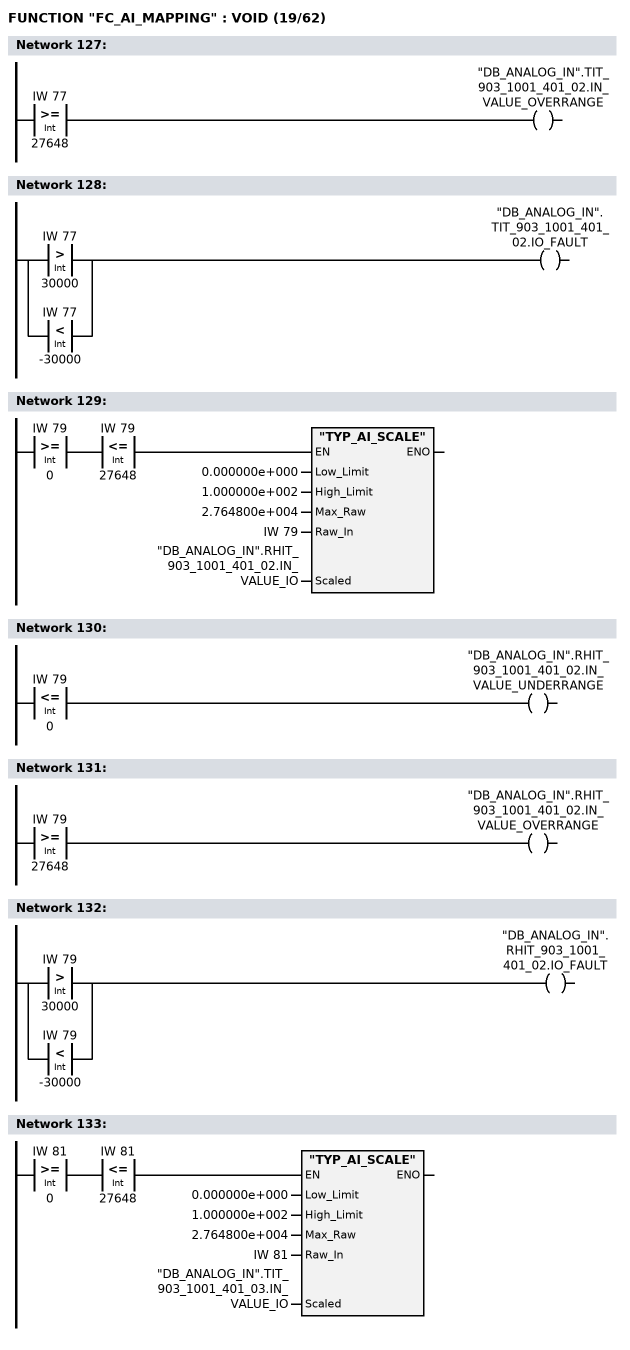

      L     IW      77;
      L     27648;
      >=I   ;
      =     "DB_ANALOG_IN".TIT_903_1001_401_02.IN_VALUE_OVERRANGE;
NETWORK
TITLE =

      O(    ;
      L     IW      77;
      L     30000;
      >I    ;
      )     ;
      O(    ;
      L     IW      77;
      L     -30000;
      <I    ;
      )     ;
      =     "DB_ANALOG_IN".TIT_903_1001_401_02.IO_FAULT;

NETWORK
TITLE =

      A(    ;
      L     IW      79;
      L     0;
      >=I   ;
      )     ;
      A(    ;
      L     IW      79;

      L     27648;
      <=I   ;
      )     ;
      JNB   _021;
      CALL "TYP_AI_SCALE" (
           Low_Limit                := 0.000000e+000,
           High_Limit               := 1.000000e+002,
           Max_Raw                  := 2.764800e+004,
           Raw_In                   := IW      79,
           Scaled                   := "DB_ANALOG_IN".RHIT_903_1001_401_02.IN_VALUE_IO);
_021: NOP   0;
NETWORK
TITLE =

      L     IW      79;
      L     0;
      <=I   ;
      =     "DB_ANALOG_IN".RHIT_903_1001_401_02.IN_VALUE_UNDERRANGE;
NETWORK
TITLE =

      L     IW      79;
      L     27648;
      >=I   ;
      =     "DB_ANALOG_IN".RHIT_903_1001_401_02.IN_VALUE_OVERRANGE;
NETWORK
TITLE =

      O(    ;
      L     IW      79;
      L     30000;
      >I    ;
      )     ;
      O(    ;
      L     IW      79;
      L     -30000;
      <I    ;
      )     ;
      =     "DB_ANALOG_IN".RHIT_903_1001_401_02.IO_FAULT;

NETWORK
TITLE =

      A(    ;
      L     IW      81;
      L     0;
      >=I   ;
      )     ;
      A(    ;
      L     IW      81;

      L     27648;
      <=I   ;
      )     ;
      JNB   _022;
      CALL "TYP_AI_SCALE" (
           Low_Limit                := 0.000000e+000,
           High_Limit               := 1.000000e+002,
           Max_Raw                  := 2.764800e+004,
           Raw_In                   := IW      81,
           Scaled                   := "DB_ANALOG_IN".TIT_903_1001_401_03.IN_VALUE_IO);
_022: NOP   0;
NETWORK
TITLE =
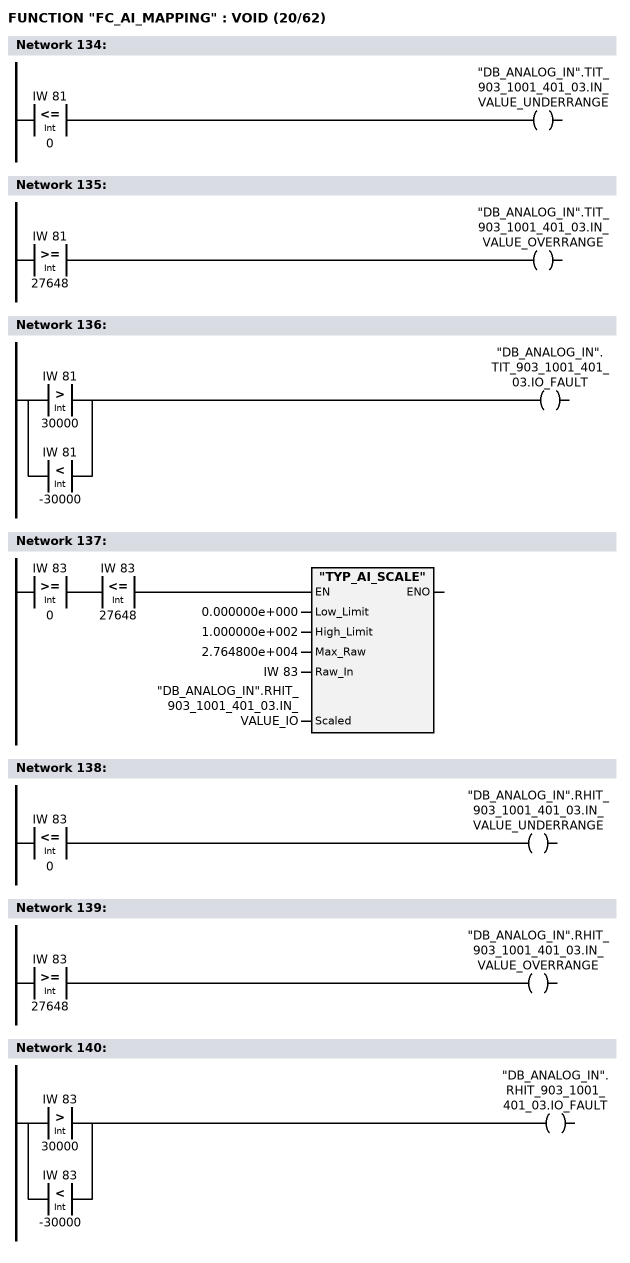

      L     IW      81;
      L     0;
      <=I   ;
      =     "DB_ANALOG_IN".TIT_903_1001_401_03.IN_VALUE_UNDERRANGE;
NETWORK
TITLE =

      L     IW      81;
      L     27648;
      >=I   ;
      =     "DB_ANALOG_IN".TIT_903_1001_401_03.IN_VALUE_OVERRANGE;
NETWORK
TITLE =

      O(    ;
      L     IW      81;
      L     30000;
      >I    ;
      )     ;
      O(    ;
      L     IW      81;
      L     -30000;
      <I    ;
      )     ;
      =     "DB_ANALOG_IN".TIT_903_1001_401_03.IO_FAULT;

NETWORK
TITLE =

      A(    ;
      L     IW      83;
      L     0;
      >=I   ;
      )     ;
      A(    ;
      L     IW      83;

      L     27648;
      <=I   ;
      )     ;
      JNB   _023;
      CALL "TYP_AI_SCALE" (
           Low_Limit                := 0.000000e+000,
           High_Limit               := 1.000000e+002,
           Max_Raw                  := 2.764800e+004,
           Raw_In                   := IW      83,
           Scaled                   := "DB_ANALOG_IN".RHIT_903_1001_401_03.IN_VALUE_IO);
_023: NOP   0;
NETWORK
TITLE =

      L     IW      83;
      L     0;
      <=I   ;
      =     "DB_ANALOG_IN".RHIT_903_1001_401_03.IN_VALUE_UNDERRANGE;
NETWORK
TITLE =

      L     IW      83;
      L     27648;
      >=I   ;
      =     "DB_ANALOG_IN".RHIT_903_1001_401_03.IN_VALUE_OVERRANGE;
NETWORK
TITLE =

      O(    ;
      L     IW      83;
      L     30000;
      >I    ;
      )     ;
      O(    ;
      L     IW      83;
      L     -30000;
      <I    ;
      )     ;
      =     "DB_ANALOG_IN".RHIT_903_1001_401_03.IO_FAULT;

NETWORK
TITLE =
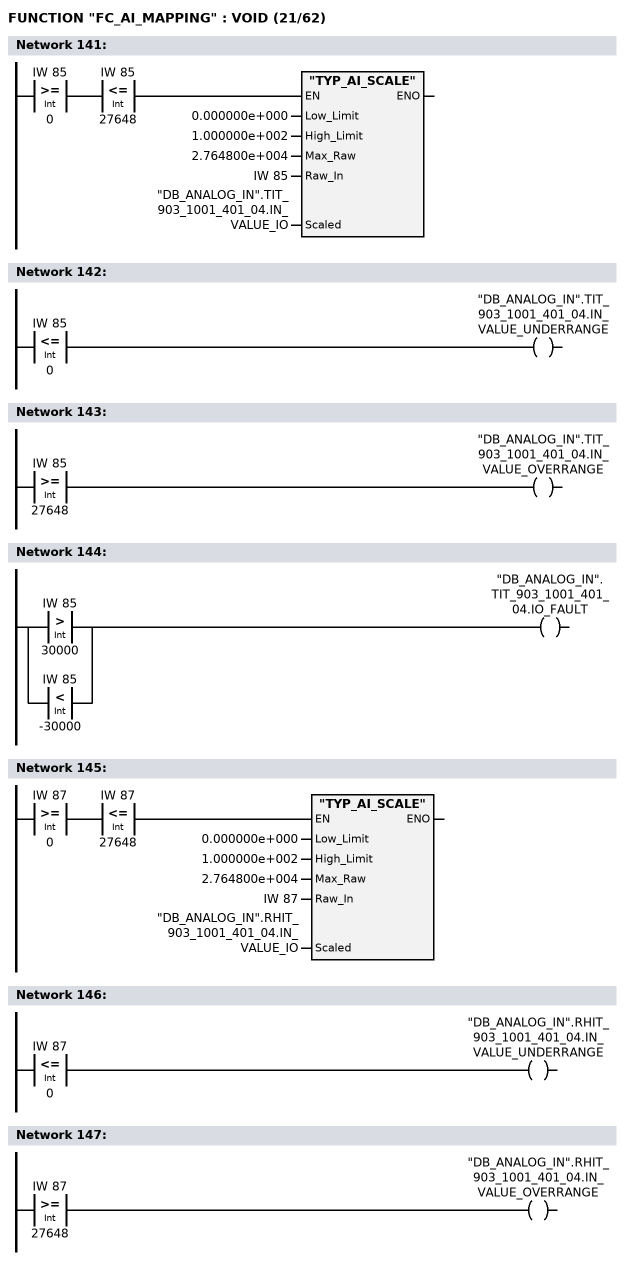

      A(    ;
      L     IW      85;
      L     0;
      >=I   ;
      )     ;
      A(    ;
      L     IW      85;

      L     27648;
      <=I   ;
      )     ;
      JNB   _024;
      CALL "TYP_AI_SCALE" (
           Low_Limit                := 0.000000e+000,
           High_Limit               := 1.000000e+002,
           Max_Raw                  := 2.764800e+004,
           Raw_In                   := IW      85,
           Scaled                   := "DB_ANALOG_IN".TIT_903_1001_401_04.IN_VALUE_IO);
_024: NOP   0;
NETWORK
TITLE =

      L     IW      85;
      L     0;
      <=I   ;
      =     "DB_ANALOG_IN".TIT_903_1001_401_04.IN_VALUE_UNDERRANGE;
NETWORK
TITLE =

      L     IW      85;
      L     27648;
      >=I   ;
      =     "DB_ANALOG_IN".TIT_903_1001_401_04.IN_VALUE_OVERRANGE;
NETWORK
TITLE =

      O(    ;
      L     IW      85;
      L     30000;
      >I    ;
      )     ;
      O(    ;
      L     IW      85;
      L     -30000;
      <I    ;
      )     ;
      =     "DB_ANALOG_IN".TIT_903_1001_401_04.IO_FAULT;

NETWORK
TITLE =

      A(    ;
      L     IW      87;
      L     0;
      >=I   ;
      )     ;
      A(    ;
      L     IW      87;

      L     27648;
      <=I   ;
      )     ;
      JNB   _025;
      CALL "TYP_AI_SCALE" (
           Low_Limit                := 0.000000e+000,
           High_Limit               := 1.000000e+002,
           Max_Raw                  := 2.764800e+004,
           Raw_In                   := IW      87,
           Scaled                   := "DB_ANALOG_IN".RHIT_903_1001_401_04.IN_VALUE_IO);
_025: NOP   0;
NETWORK
TITLE =

      L     IW      87;
      L     0;
      <=I   ;
      =     "DB_ANALOG_IN".RHIT_903_1001_401_04.IN_VALUE_UNDERRANGE;
NETWORK
TITLE =

      L     IW      87;
      L     27648;
      >=I   ;
      =     "DB_ANALOG_IN".RHIT_903_1001_401_04.IN_VALUE_OVERRANGE;
NETWORK
TITLE =
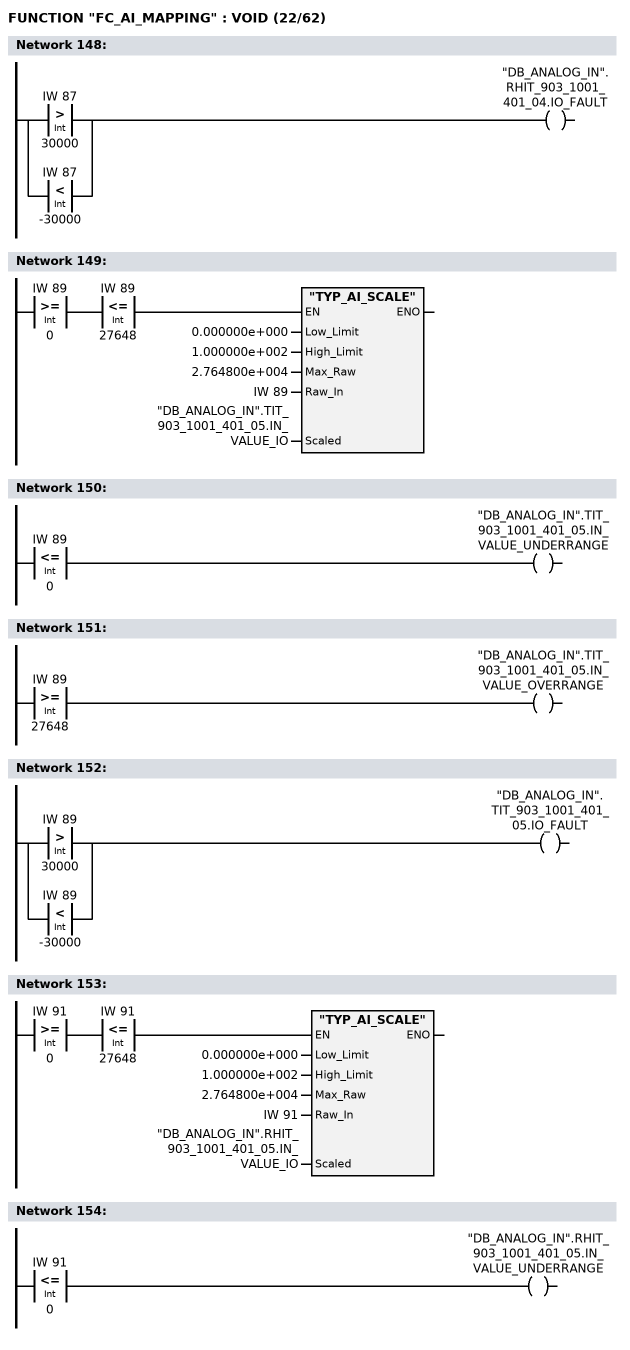

      O(    ;
      L     IW      87;
      L     30000;
      >I    ;
      )     ;
      O(    ;
      L     IW      87;
      L     -30000;
      <I    ;
      )     ;
      =     "DB_ANALOG_IN".RHIT_903_1001_401_04.IO_FAULT;

NETWORK
TITLE =

      A(    ;
      L     IW      89;
      L     0;
      >=I   ;
      )     ;
      A(    ;
      L     IW      89;

      L     27648;
      <=I   ;
      )     ;
      JNB   _026;
      CALL "TYP_AI_SCALE" (
           Low_Limit                := 0.000000e+000,
           High_Limit               := 1.000000e+002,
           Max_Raw                  := 2.764800e+004,
           Raw_In                   := IW      89,
           Scaled                   := "DB_ANALOG_IN".TIT_903_1001_401_05.IN_VALUE_IO);
_026: NOP   0;
NETWORK
TITLE =

      L     IW      89;
      L     0;
      <=I   ;
      =     "DB_ANALOG_IN".TIT_903_1001_401_05.IN_VALUE_UNDERRANGE;
NETWORK
TITLE =

      L     IW      89;
      L     27648;
      >=I   ;
      =     "DB_ANALOG_IN".TIT_903_1001_401_05.IN_VALUE_OVERRANGE;
NETWORK
TITLE =

      O(    ;
      L     IW      89;
      L     30000;
      >I    ;
      )     ;
      O(    ;
      L     IW      89;
      L     -30000;
      <I    ;
      )     ;
      =     "DB_ANALOG_IN".TIT_903_1001_401_05.IO_FAULT;

NETWORK
TITLE =

      A(    ;
      L     IW      91;
      L     0;
      >=I   ;
      )     ;
      A(    ;
      L     IW      91;

      L     27648;
      <=I   ;
      )     ;
      JNB   _027;
      CALL "TYP_AI_SCALE" (
           Low_Limit                := 0.000000e+000,
           High_Limit               := 1.000000e+002,
           Max_Raw                  := 2.764800e+004,
           Raw_In                   := IW      91,
           Scaled                   := "DB_ANALOG_IN".RHIT_903_1001_401_05.IN_VALUE_IO);
_027: NOP   0;
NETWORK
TITLE =

      L     IW      91;
      L     0;
      <=I   ;
      =     "DB_ANALOG_IN".RHIT_903_1001_401_05.IN_VALUE_UNDERRANGE;
NETWORK
TITLE =
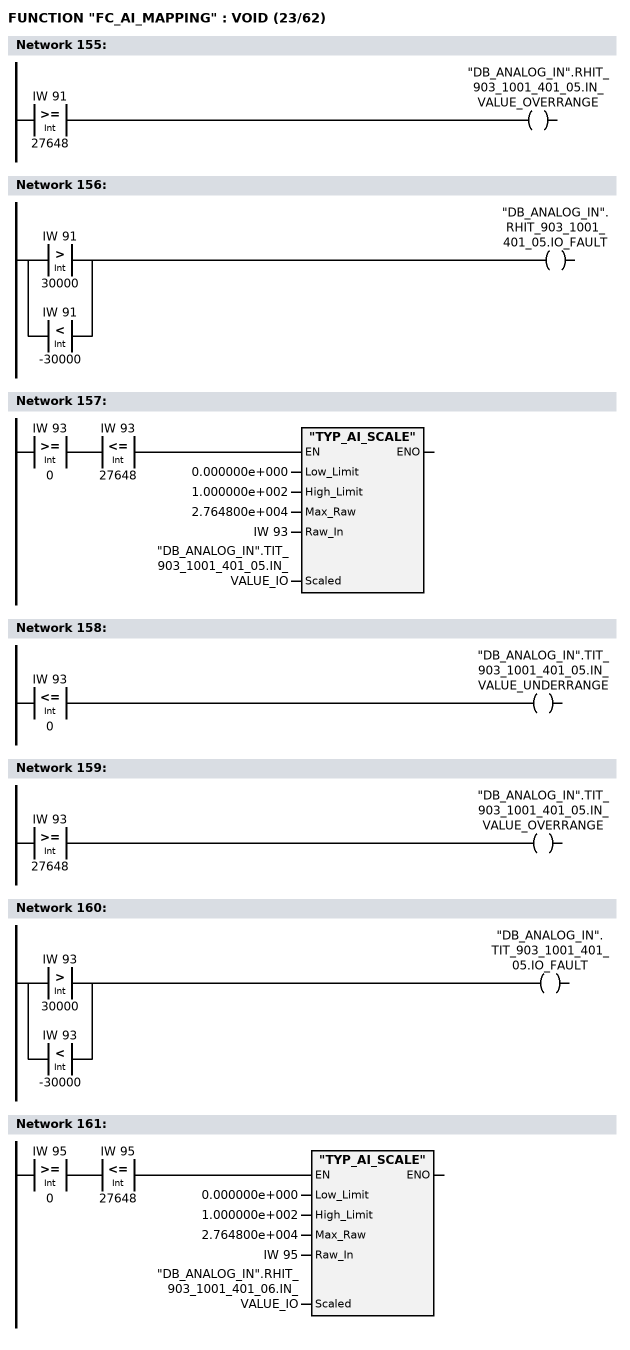

      L     IW      91;
      L     27648;
      >=I   ;
      =     "DB_ANALOG_IN".RHIT_903_1001_401_05.IN_VALUE_OVERRANGE;
NETWORK
TITLE =

      O(    ;
      L     IW      91;
      L     30000;
      >I    ;
      )     ;
      O(    ;
      L     IW      91;
      L     -30000;
      <I    ;
      )     ;
      =     "DB_ANALOG_IN".RHIT_903_1001_401_05.IO_FAULT;

NETWORK
TITLE =

      A(    ;
      L     IW      93;
      L     0;
      >=I   ;
      )     ;
      A(    ;
      L     IW      93;

      L     27648;
      <=I   ;
      )     ;
      JNB   _028;
      CALL "TYP_AI_SCALE" (
           Low_Limit                := 0.000000e+000,
           High_Limit               := 1.000000e+002,
           Max_Raw                  := 2.764800e+004,
           Raw_In                   := IW      93,
           Scaled                   := "DB_ANALOG_IN".TIT_903_1001_401_05.IN_VALUE_IO);
_028: NOP   0;
NETWORK
TITLE =

      L     IW      93;
      L     0;
      <=I   ;
      =     "DB_ANALOG_IN".TIT_903_1001_401_05.IN_VALUE_UNDERRANGE;
NETWORK
TITLE =

      L     IW      93;
      L     27648;
      >=I   ;
      =     "DB_ANALOG_IN".TIT_903_1001_401_05.IN_VALUE_OVERRANGE;
NETWORK
TITLE =

      O(    ;
      L     IW      93;
      L     30000;
      >I    ;
      )     ;
      O(    ;
      L     IW      93;
      L     -30000;
      <I    ;
      )     ;
      =     "DB_ANALOG_IN".TIT_903_1001_401_05.IO_FAULT;

NETWORK
TITLE =

      A(    ;
      L     IW      95;
      L     0;
      >=I   ;
      )     ;
      A(    ;
      L     IW      95;

      L     27648;
      <=I   ;
      )     ;
      JNB   _029;
      CALL "TYP_AI_SCALE" (
           Low_Limit                := 0.000000e+000,
           High_Limit               := 1.000000e+002,
           Max_Raw                  := 2.764800e+004,
           Raw_In                   := IW      95,
           Scaled                   := "DB_ANALOG_IN".RHIT_903_1001_401_06.IN_VALUE_IO);
_029: NOP   0;
NETWORK
TITLE =
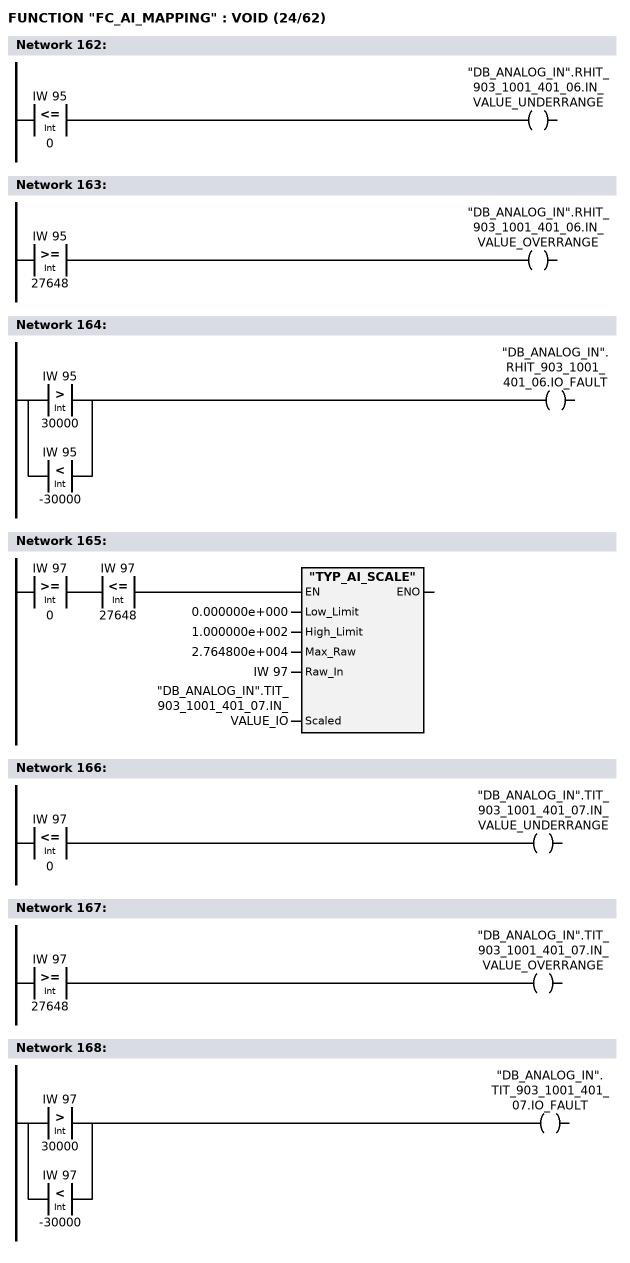

      L     IW      95;
      L     0;
      <=I   ;
      =     "DB_ANALOG_IN".RHIT_903_1001_401_06.IN_VALUE_UNDERRANGE;
NETWORK
TITLE =

      L     IW      95;
      L     27648;
      >=I   ;
      =     "DB_ANALOG_IN".RHIT_903_1001_401_06.IN_VALUE_OVERRANGE;
NETWORK
TITLE =

      O(    ;
      L     IW      95;
      L     30000;
      >I    ;
      )     ;
      O(    ;
      L     IW      95;
      L     -30000;
      <I    ;
      )     ;
      =     "DB_ANALOG_IN".RHIT_903_1001_401_06.IO_FAULT;

NETWORK
TITLE =

      A(    ;
      L     IW      97;
      L     0;
      >=I   ;
      )     ;
      A(    ;
      L     IW      97;

      L     27648;
      <=I   ;
      )     ;
      JNB   _02a;
      CALL "TYP_AI_SCALE" (
           Low_Limit                := 0.000000e+000,
           High_Limit               := 1.000000e+002,
           Max_Raw                  := 2.764800e+004,
           Raw_In                   := IW      97,
           Scaled                   := "DB_ANALOG_IN".TIT_903_1001_401_07.IN_VALUE_IO);
_02a: NOP   0;
NETWORK
TITLE =

      L     IW      97;
      L     0;
      <=I   ;
      =     "DB_ANALOG_IN".TIT_903_1001_401_07.IN_VALUE_UNDERRANGE;
NETWORK
TITLE =

      L     IW      97;
      L     27648;
      >=I   ;
      =     "DB_ANALOG_IN".TIT_903_1001_401_07.IN_VALUE_OVERRANGE;
NETWORK
TITLE =

      O(    ;
      L     IW      97;
      L     30000;
      >I    ;
      )     ;
      O(    ;
      L     IW      97;
      L     -30000;
      <I    ;
      )     ;
      =     "DB_ANALOG_IN".TIT_903_1001_401_07.IO_FAULT;

NETWORK
TITLE =
